REGION Network 54: CM Vision Z Axis Command posAbsolute
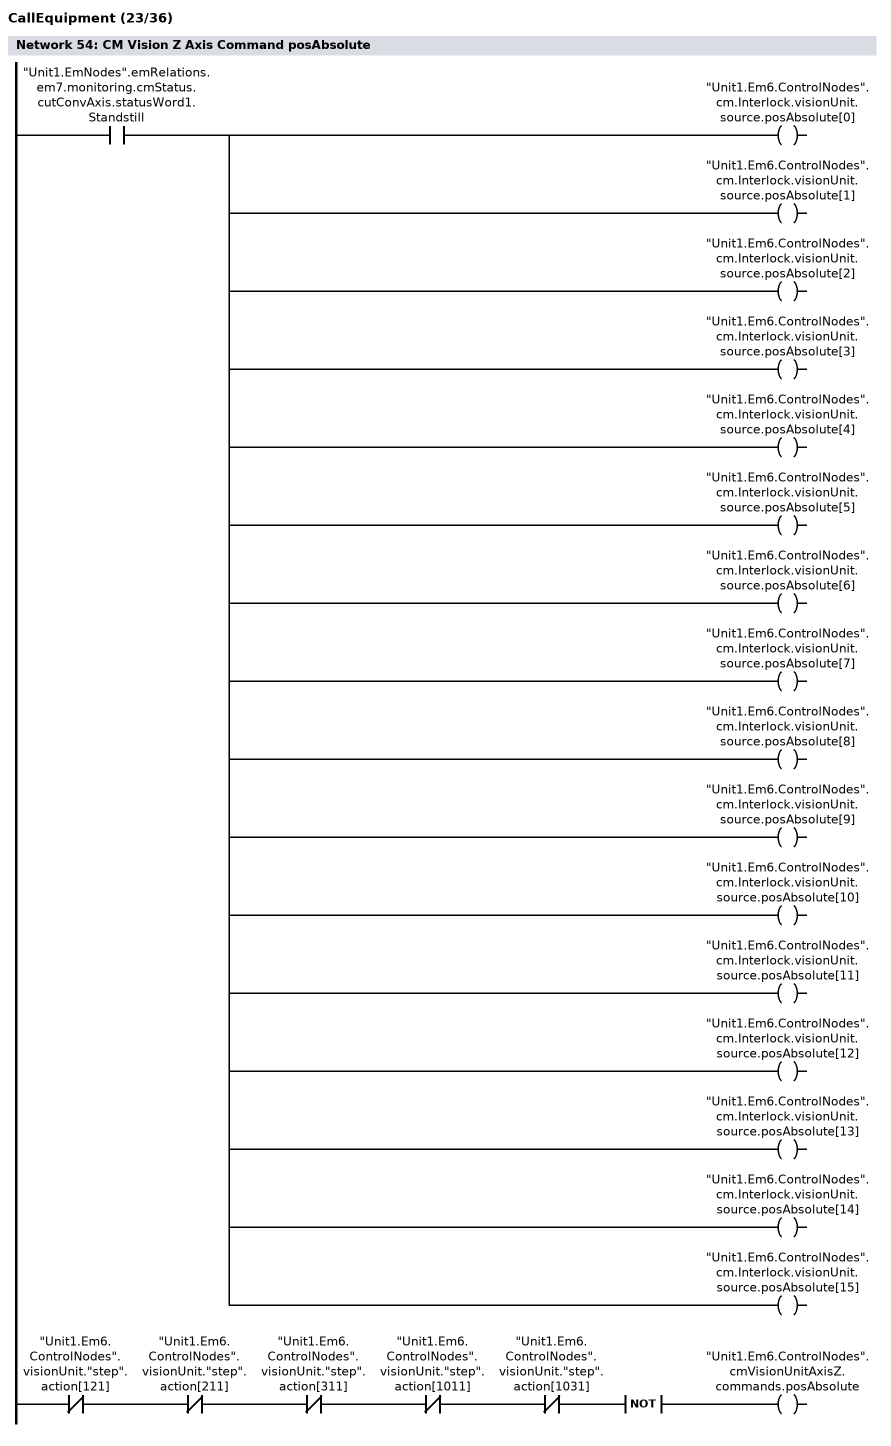
   RUNG wire#powerrail
      Contact( "Unit1.EmNodes".emRelations.em7.monitoring.cmStatus.cutConvAxis.statusWord1.Standstill )
      wire#w1
      Coil( "Unit1.Em6.ControlNodes".cm.Interlock.visionUnit.source.posAbsolute[0] )
   END_RUNG
   RUNG wire#w1
      Coil( "Unit1.Em6.ControlNodes".cm.Interlock.visionUnit.source.posAbsolute[1] )
   END_RUNG
   RUNG wire#w1
      Coil( "Unit1.Em6.ControlNodes".cm.Interlock.visionUnit.source.posAbsolute[2] )
   END_RUNG
   RUNG wire#w1
      Coil( "Unit1.Em6.ControlNodes".cm.Interlock.visionUnit.source.posAbsolute[3] )
   END_RUNG
   RUNG wire#w1
      Coil( "Unit1.Em6.ControlNodes".cm.Interlock.visionUnit.source.posAbsolute[4] )
   END_RUNG
   RUNG wire#w1
      Coil( "Unit1.Em6.ControlNodes".cm.Interlock.visionUnit.source.posAbsolute[5] )
   END_RUNG
   RUNG wire#w1
      Coil( "Unit1.Em6.ControlNodes".cm.Interlock.visionUnit.source.posAbsolute[6] )
   END_RUNG
   RUNG wire#w1
      Coil( "Unit1.Em6.ControlNodes".cm.Interlock.visionUnit.source.posAbsolute[7] )
   END_RUNG
   RUNG wire#w1
      Coil( "Unit1.Em6.ControlNodes".cm.Interlock.visionUnit.source.posAbsolute[8] )
   END_RUNG
   RUNG wire#w1
      Coil( "Unit1.Em6.ControlNodes".cm.Interlock.visionUnit.source.posAbsolute[9] )
   END_RUNG
   RUNG wire#w1
      Coil( "Unit1.Em6.ControlNodes".cm.Interlock.visionUnit.source.posAbsolute[10] )
   END_RUNG
   RUNG wire#w1
      Coil( "Unit1.Em6.ControlNodes".cm.Interlock.visionUnit.source.posAbsolute[11] )
   END_RUNG
   RUNG wire#w1
      Coil( "Unit1.Em6.ControlNodes".cm.Interlock.visionUnit.source.posAbsolute[12] )
   END_RUNG
   RUNG wire#w1
      Coil( "Unit1.Em6.ControlNodes".cm.Interlock.visionUnit.source.posAbsolute[13] )
   END_RUNG
   RUNG wire#w1
      Coil( "Unit1.Em6.ControlNodes".cm.Interlock.visionUnit.source.posAbsolute[14] )
   END_RUNG
   RUNG wire#w1
      Coil( "Unit1.Em6.ControlNodes".cm.Interlock.visionUnit.source.posAbsolute[15] )
   END_RUNG
   RUNG wire#powerrail
      I_Contact( "Unit1.Em6.ControlNodes".visionUnit."step".action[121] )
      I_Contact( "Unit1.Em6.ControlNodes".visionUnit."step".action[211] )
      I_Contact( "Unit1.Em6.ControlNodes".visionUnit."step".action[311] )
      I_Contact( "Unit1.Em6.ControlNodes".visionUnit."step".action[1011] )
      I_Contact( "Unit1.Em6.ControlNodes".visionUnit."step".action[1031] )
      Not()
      Coil( "Unit1.Em6.ControlNodes".cmVisionUnitAxisZ.commands.posAbsolute )
   END_RUNG
   // the same network as SCL:
   "Unit1.Em6.ControlNodes".cm.Interlock.visionUnit.source.posAbsolute[0] := "Unit1.EmNodes".emRelations.em7.monitoring.cmStatus.cutConvAxis.statusWord1.Standstill;
   "Unit1.Em6.ControlNodes".cm.Interlock.visionUnit.source.posAbsolute[1] := "Unit1.EmNodes".emRelations.em7.monitoring.cmStatus.cutConvAxis.statusWord1.Standstill;
   "Unit1.Em6.ControlNodes".cm.Interlock.visionUnit.source.posAbsolute[2] := "Unit1.EmNodes".emRelations.em7.monitoring.cmStatus.cutConvAxis.statusWord1.Standstill;
   "Unit1.Em6.ControlNodes".cm.Interlock.visionUnit.source.posAbsolute[3] := "Unit1.EmNodes".emRelations.em7.monitoring.cmStatus.cutConvAxis.statusWord1.Standstill;
   "Unit1.Em6.ControlNodes".cm.Interlock.visionUnit.source.posAbsolute[4] := "Unit1.EmNodes".emRelations.em7.monitoring.cmStatus.cutConvAxis.statusWord1.Standstill;
   "Unit1.Em6.ControlNodes".cm.Interlock.visionUnit.source.posAbsolute[5] := "Unit1.EmNodes".emRelations.em7.monitoring.cmStatus.cutConvAxis.statusWord1.Standstill;
   "Unit1.Em6.ControlNodes".cm.Interlock.visionUnit.source.posAbsolute[6] := "Unit1.EmNodes".emRelations.em7.monitoring.cmStatus.cutConvAxis.statusWord1.Standstill;
   "Unit1.Em6.ControlNodes".cm.Interlock.visionUnit.source.posAbsolute[7] := "Unit1.EmNodes".emRelations.em7.monitoring.cmStatus.cutConvAxis.statusWord1.Standstill;
   "Unit1.Em6.ControlNodes".cm.Interlock.visionUnit.source.posAbsolute[8] := "Unit1.EmNodes".emRelations.em7.monitoring.cmStatus.cutConvAxis.statusWord1.Standstill;
   "Unit1.Em6.ControlNodes".cm.Interlock.visionUnit.source.posAbsolute[9] := "Unit1.EmNodes".emRelations.em7.monitoring.cmStatus.cutConvAxis.statusWord1.Standstill;
   "Unit1.Em6.ControlNodes".cm.Interlock.visionUnit.source.posAbsolute[10] := "Unit1.EmNodes".emRelations.em7.monitoring.cmStatus.cutConvAxis.statusWord1.Standstill;
   "Unit1.Em6.ControlNodes".cm.Interlock.visionUnit.source.posAbsolute[11] := "Unit1.EmNodes".emRelations.em7.monitoring.cmStatus.cutConvAxis.statusWord1.Standstill;
   "Unit1.Em6.ControlNodes".cm.Interlock.visionUnit.source.posAbsolute[12] := "Unit1.EmNodes".emRelations.em7.monitoring.cmStatus.cutConvAxis.statusWord1.Standstill;
   "Unit1.Em6.ControlNodes".cm.Interlock.visionUnit.source.posAbsolute[13] := "Unit1.EmNodes".emRelations.em7.monitoring.cmStatus.cutConvAxis.statusWord1.Standstill;
   "Unit1.Em6.ControlNodes".cm.Interlock.visionUnit.source.posAbsolute[14] := "Unit1.EmNodes".emRelations.em7.monitoring.cmStatus.cutConvAxis.statusWord1.Standstill;
   "Unit1.Em6.ControlNodes".cm.Interlock.visionUnit.source.posAbsolute[15] := "Unit1.EmNodes".emRelations.em7.monitoring.cmStatus.cutConvAxis.statusWord1.Standstill;
   "Unit1.Em6.ControlNodes".cmVisionUnitAxisZ.commands.posAbsolute := NOT (NOT "Unit1.Em6.ControlNodes".visionUnit."step".action[121] AND NOT "Unit1.Em6.ControlNodes".visionUnit."step".action[211] AND NOT "Unit1.Em6.ControlNodes".visionUnit."step".action[311] AND NOT "Unit1.Em6.ControlNodes".visionUnit."step".action[1011] AND NOT "Unit1.Em6.ControlNodes".visionUnit."step".action[1031]);
END_REGION

REGION Network 55: Call CM Vision Z Axis (LER_Interlock Summary)
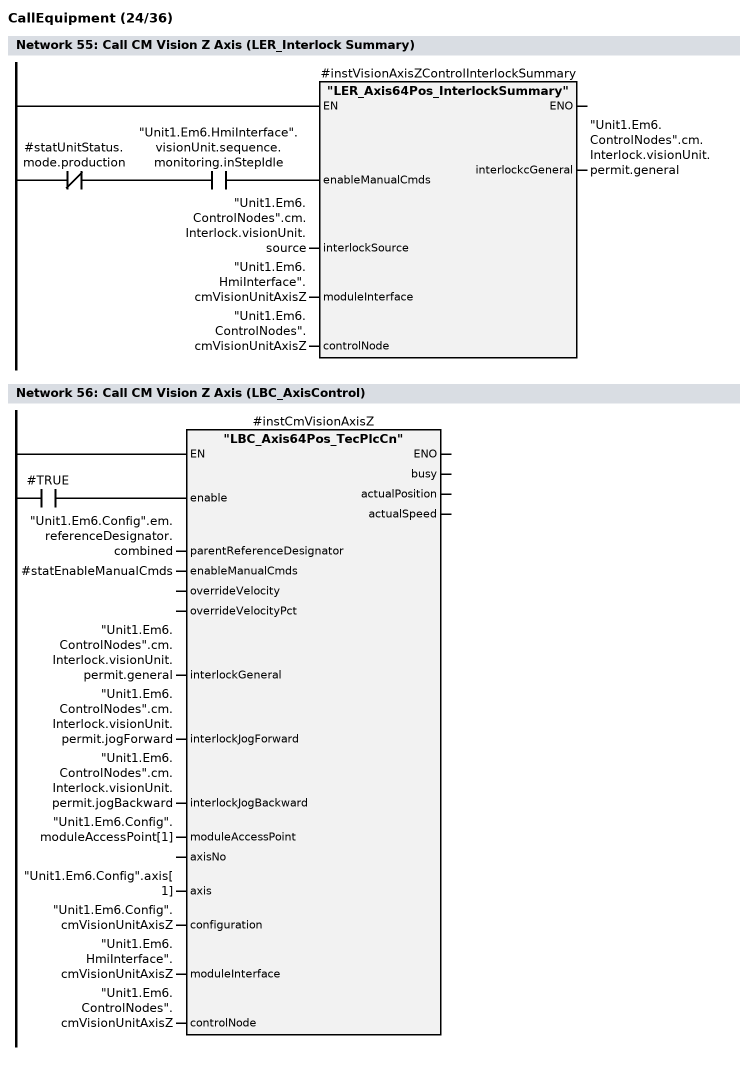
   RUNG wire#powerrail
      #instVisionAxisZControlInterlockSummary(enableManualCmds := wire#w1, interlockSource := "Unit1.Em6.ControlNodes".cm.Interlock.visionUnit.source, moduleInterface := "Unit1.Em6.HmiInterface".cmVisionUnitAxisZ, controlNode := "Unit1.Em6.ControlNodes".cmVisionUnitAxisZ, interlockcGeneral => "Unit1.Em6.ControlNodes".cm.Interlock.visionUnit.permit.general)
   END_RUNG
   RUNG wire#powerrail
      I_Contact( #statUnitStatus.mode.production )
      Contact( "Unit1.Em6.HmiInterface".visionUnit.sequence.monitoring.inStepIdle )
   END_RUNG wire#w1
   // the same network as SCL:
   #instVisionAxisZControlInterlockSummary(enableManualCmds := NOT #statUnitStatus.mode.production AND "Unit1.Em6.HmiInterface".visionUnit.sequence.monitoring.inStepIdle,   // "LER_Axis64Pos_InterlockSummary"
                           interlockSource := "Unit1.Em6.ControlNodes".cm.Interlock.visionUnit.source,
                           moduleInterface := "Unit1.Em6.HmiInterface".cmVisionUnitAxisZ,
                           controlNode := "Unit1.Em6.ControlNodes".cmVisionUnitAxisZ,
                           interlockcGeneral => "Unit1.Em6.ControlNodes".cm.Interlock.visionUnit.permit.general);
END_REGION

REGION Network 56: Call CM Vision Z Axis (LBC_AxisControl)
   RUNG wire#powerrail
      #instCmVisionAxisZ(enable := wire#w1, parentReferenceDesignator := "Unit1.Em6.Config".em.referenceDesignator.combined, enableManualCmds := #statEnableManualCmds, overrideVelocity :=, overrideVelocityPct :=, interlockGeneral := "Unit1.Em6.ControlNodes".cm.Interlock.visionUnit.permit.general, interlockJogForward := "Unit1.Em6.ControlNodes".cm.Interlock.visionUnit.permit.jogForward, interlockJogBackward := "Unit1.Em6.ControlNodes".cm.Interlock.visionUnit.permit.jogBackward, moduleAccessPoint := "Unit1.Em6.Config".moduleAccessPoint[1], axisNo :=, axis := "Unit1.Em6.Config".axis[1], configuration := "Unit1.Em6.Config".cmVisionUnitAxisZ, moduleInterface := "Unit1.Em6.HmiInterface".cmVisionUnitAxisZ, controlNode := "Unit1.Em6.ControlNodes".cmVisionUnitAxisZ, busy =>, actualPosition =>, actualSpeed =>)
   END_RUNG
   RUNG wire#powerrail
      Contact( #TRUE )
   END_RUNG wire#w1
   // the same network as SCL:
   #instCmVisionAxisZ(enable := #TRUE,   // "LBC_Axis64Pos_TecPlcCn"
                      parentReferenceDesignator := "Unit1.Em6.Config".em.referenceDesignator.combined,
                      enableManualCmds := #statEnableManualCmds,
                      interlockGeneral := "Unit1.Em6.ControlNodes".cm.Interlock.visionUnit.permit.general,
                      interlockJogForward := "Unit1.Em6.ControlNodes".cm.Interlock.visionUnit.permit.jogForward,
                      interlockJogBackward := "Unit1.Em6.ControlNodes".cm.Interlock.visionUnit.permit.jogBackward,
                      moduleAccessPoint := "Unit1.Em6.Config".moduleAccessPoint[1],
                      axis := "Unit1.Em6.Config".axis[1],
                      configuration := "Unit1.Em6.Config".cmVisionUnitAxisZ,
                      moduleInterface := "Unit1.Em6.HmiInterface".cmVisionUnitAxisZ,
                      controlNode := "Unit1.Em6.ControlNodes".cmVisionUnitAxisZ);
END_REGION

REGION Network 57: Call CM Vision Z Axis (LER_ServoTorqueCal)
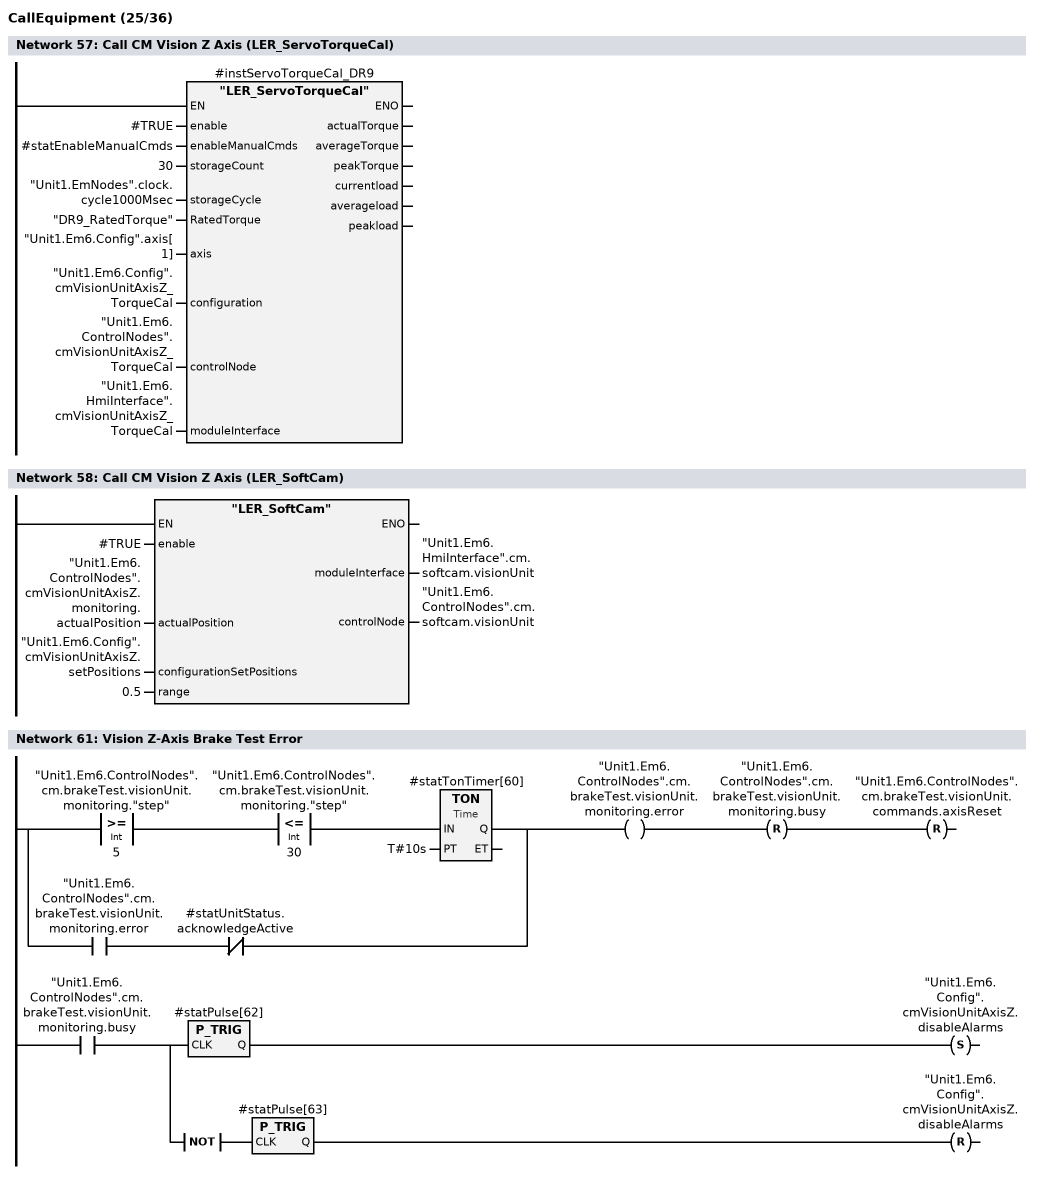
   RUNG wire#powerrail
      #instServoTorqueCal_DR9(enable := #TRUE, enableManualCmds := #statEnableManualCmds, storageCount := 30, storageCycle := "Unit1.EmNodes".clock.cycle1000Msec, RatedTorque := "DR9_RatedTorque", axis := "Unit1.Em6.Config".axis[1], configuration := "Unit1.Em6.Config".cmVisionUnitAxisZ_TorqueCal, controlNode := "Unit1.Em6.ControlNodes".cmVisionUnitAxisZ_TorqueCal, moduleInterface := "Unit1.Em6.HmiInterface".cmVisionUnitAxisZ_TorqueCal, actualTorque =>, averageTorque =>, peakTorque =>, currentload =>, averageload =>, peakload =>)
   END_RUNG
   // the same network as SCL:
   #instServoTorqueCal_DR9(enable := #TRUE,   // "LER_ServoTorqueCal"
                           enableManualCmds := #statEnableManualCmds,
                           storageCount := 30,
                           storageCycle := "Unit1.EmNodes".clock.cycle1000Msec,
                           RatedTorque := "DR9_RatedTorque",
                           axis := "Unit1.Em6.Config".axis[1],
                           configuration := "Unit1.Em6.Config".cmVisionUnitAxisZ_TorqueCal,
                           controlNode := "Unit1.Em6.ControlNodes".cmVisionUnitAxisZ_TorqueCal,
                           moduleInterface := "Unit1.Em6.HmiInterface".cmVisionUnitAxisZ_TorqueCal);
END_REGION

REGION Network 58: Call CM Vision Z Axis (LER_SoftCam)
   RUNG wire#powerrail
      "LER_SoftCam"(enable := #TRUE, actualPosition := "Unit1.Em6.ControlNodes".cmVisionUnitAxisZ.monitoring.actualPosition, configurationSetPositions := "Unit1.Em6.Config".cmVisionUnitAxisZ.setPositions, range := 0.5, moduleInterface => "Unit1.Em6.HmiInterface".cm.softcam.visionUnit, controlNode => "Unit1.Em6.ControlNodes".cm.softcam.visionUnit)
   END_RUNG
   // the same network as SCL:
   "LER_SoftCam"(enable := #TRUE,
                 actualPosition := "Unit1.Em6.ControlNodes".cmVisionUnitAxisZ.monitoring.actualPosition,
                 configurationSetPositions := "Unit1.Em6.Config".cmVisionUnitAxisZ.setPositions,
                 range := 0.5,
                 moduleInterface => "Unit1.Em6.HmiInterface".cm.softcam.visionUnit,
                 controlNode => "Unit1.Em6.ControlNodes".cm.softcam.visionUnit);
END_REGION

REGION Network 60: ******************** Brake Test (Axis) ********************
END_REGION

REGION Network 61: Vision Z-Axis Brake Test Error
   RUNG wire#powerrail
      { S7_Templates := "SrcType := Int" } GE_Contact(in1 := "Unit1.Em6.ControlNodes".cm.brakeTest.visionUnit.monitoring."step", in2 := 5)
      { S7_Templates := "SrcType := Int" } LE_Contact(in1 := "Unit1.Em6.ControlNodes".cm.brakeTest.visionUnit.monitoring."step", in2 := 30)
      { S7_Templates := "time_type := Time" } #statTonTimer[60].TON(pt := T#10s, et =>)
      wire#w1
      Coil( "Unit1.Em6.ControlNodes".cm.brakeTest.visionUnit.monitoring.error )
      R_Coil( "Unit1.Em6.ControlNodes".cm.brakeTest.visionUnit.monitoring.busy )
      R_Coil( "Unit1.Em6.ControlNodes".cm.brakeTest.visionUnit.commands.axisReset )
   END_RUNG
   RUNG wire#powerrail
      Contact( "Unit1.Em6.ControlNodes".cm.brakeTest.visionUnit.monitoring.error )
      I_Contact( #statUnitStatus.acknowledgeActive )
   END_RUNG wire#w1
   RUNG wire#powerrail
      Contact( "Unit1.Em6.ControlNodes".cm.brakeTest.visionUnit.monitoring.busy )
      wire#w2
      P_Trig( #statPulse[62] )
      S_Coil( "Unit1.Em6.Config".cmVisionUnitAxisZ.disableAlarms )
   END_RUNG
   RUNG wire#w2
      Not()
      P_Trig( #statPulse[63] )
      R_Coil( "Unit1.Em6.Config".cmVisionUnitAxisZ.disableAlarms )
   END_RUNG
   // the same network as SCL:
   #statTonTimer[60].TON(IN := ("Unit1.Em6.ControlNodes".cm.brakeTest.visionUnit.monitoring."step" >= 5) AND ("Unit1.Em6.ControlNodes".cm.brakeTest.visionUnit.monitoring."step" <= 30),
                         PT := T#10s);
   "Unit1.Em6.ControlNodes".cm.brakeTest.visionUnit.monitoring.error := #statTonTimer[60].Q OR ("Unit1.Em6.ControlNodes".cm.brakeTest.visionUnit.monitoring.error AND NOT #statUnitStatus.acknowledgeActive);
   IF "Unit1.Em6.ControlNodes".cm.brakeTest.visionUnit.monitoring.error THEN
       "Unit1.Em6.ControlNodes".cm.brakeTest.visionUnit.monitoring.busy := FALSE;
       "Unit1.Em6.ControlNodes".cm.brakeTest.visionUnit.commands.axisReset := FALSE;
   END_IF;
   #_w1 := "Unit1.Em6.ControlNodes".cm.brakeTest.visionUnit.monitoring.busy AND NOT #statPulse[62];   // rising edge
   #statPulse[62] := "Unit1.Em6.ControlNodes".cm.brakeTest.visionUnit.monitoring.busy;
   IF #_w1 THEN "Unit1.Em6.Config".cmVisionUnitAxisZ.disableAlarms := TRUE; END_IF;
   #_w2 := NOT "Unit1.Em6.ControlNodes".cm.brakeTest.visionUnit.monitoring.busy AND NOT #statPulse[63];   // rising edge
   #statPulse[63] := NOT "Unit1.Em6.ControlNodes".cm.brakeTest.visionUnit.monitoring.busy;
   IF #_w2 THEN "Unit1.Em6.Config".cmVisionUnitAxisZ.disableAlarms := FALSE; END_IF;
END_REGION

REGION Network 62: Vision Z-Axis Brake Test Initialize
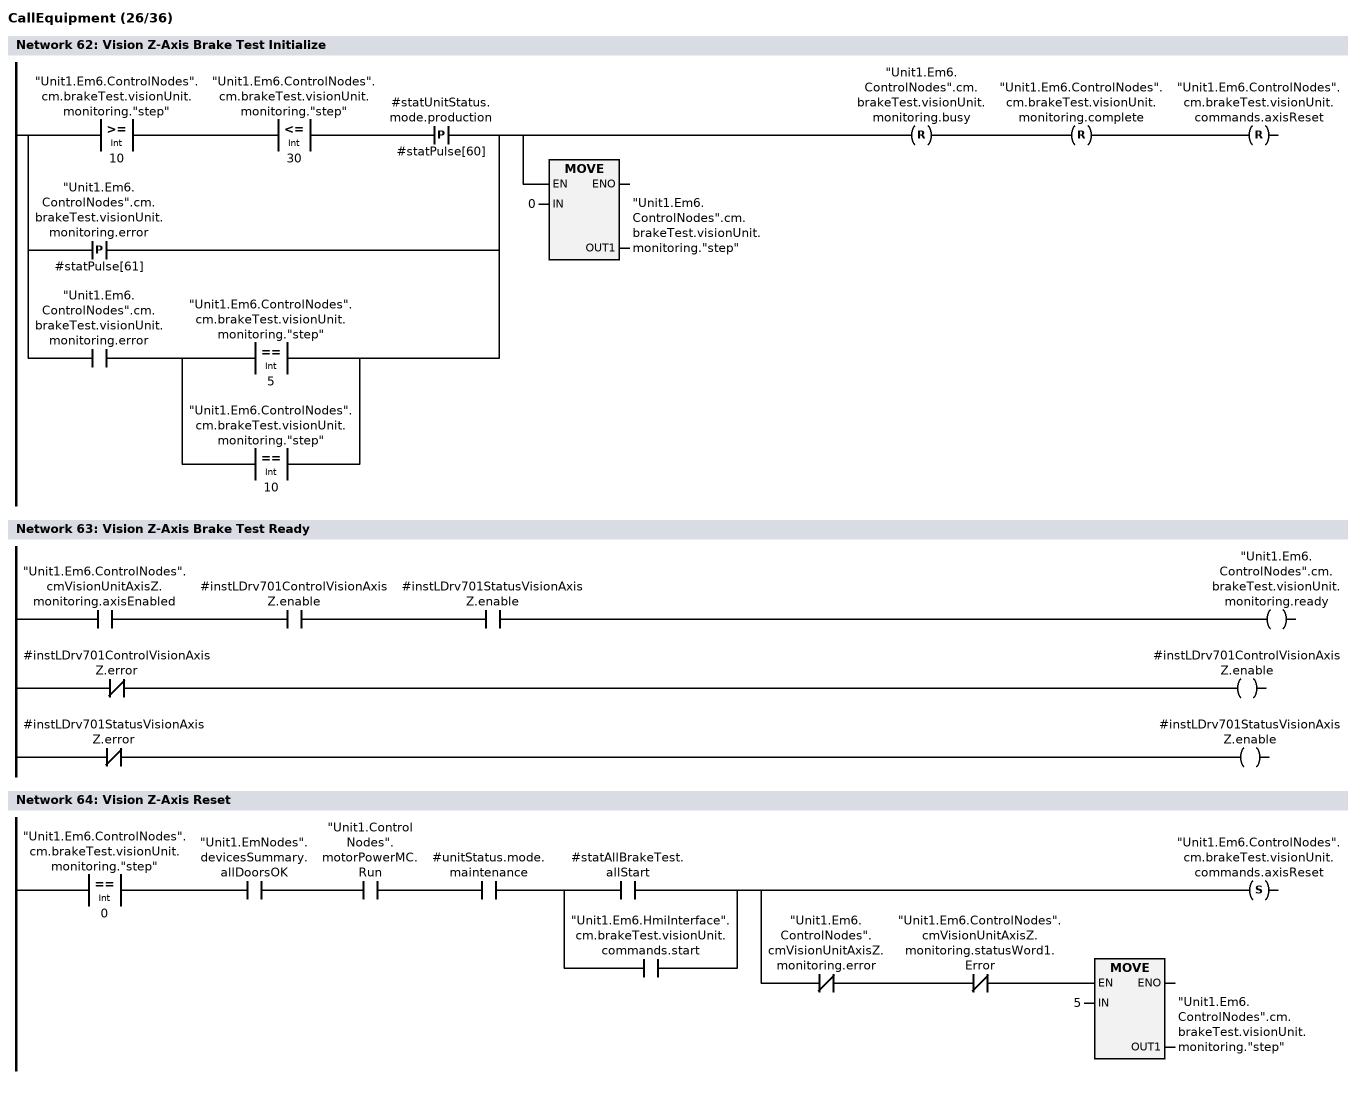
   RUNG wire#powerrail
      { S7_Templates := "SrcType := Int" } GE_Contact(in1 := "Unit1.Em6.ControlNodes".cm.brakeTest.visionUnit.monitoring."step", in2 := 10)
      { S7_Templates := "SrcType := Int" } LE_Contact(in1 := "Unit1.Em6.ControlNodes".cm.brakeTest.visionUnit.monitoring."step", in2 := 30)
      P_Contact(operand := #statUnitStatus.mode.production, bit := #statPulse[60])
      wire#w1
      R_Coil( "Unit1.Em6.ControlNodes".cm.brakeTest.visionUnit.monitoring.busy )
      R_Coil( "Unit1.Em6.ControlNodes".cm.brakeTest.visionUnit.monitoring.complete )
      R_Coil( "Unit1.Em6.ControlNodes".cm.brakeTest.visionUnit.commands.axisReset )
   END_RUNG
   RUNG wire#powerrail
      P_Contact(operand := "Unit1.Em6.ControlNodes".cm.brakeTest.visionUnit.monitoring.error, bit := #statPulse[61])
   END_RUNG wire#w1
   RUNG wire#powerrail
      Contact( "Unit1.Em6.ControlNodes".cm.brakeTest.visionUnit.monitoring.error )
      wire#w2
      { S7_Templates := "SrcType := Int" } EQ_Contact(in1 := "Unit1.Em6.ControlNodes".cm.brakeTest.visionUnit.monitoring."step", in2 := 5)
   END_RUNG wire#w1
   RUNG wire#w2
      { S7_Templates := "SrcType := Int" } EQ_Contact(in1 := "Unit1.Em6.ControlNodes".cm.brakeTest.visionUnit.monitoring."step", in2 := 10)
   END_RUNG wire#w1
   RUNG wire#w1
      Move(in := 0, out1 => "Unit1.Em6.ControlNodes".cm.brakeTest.visionUnit.monitoring."step")
   END_RUNG
   // the same network as SCL:
   #_w1 := ("Unit1.Em6.ControlNodes".cm.brakeTest.visionUnit.monitoring."step" >= 10) AND ("Unit1.Em6.ControlNodes".cm.brakeTest.visionUnit.monitoring."step" <= 30) AND #statUnitStatus.mode.production AND NOT #statPulse[60];   // rising edge of #statUnitStatus.mode.production
   #statPulse[60] := #statUnitStatus.mode.production;
   #_w2 := "Unit1.Em6.ControlNodes".cm.brakeTest.visionUnit.monitoring.error AND NOT #statPulse[61];   // rising edge of "Unit1.Em6.ControlNodes".cm.brakeTest.visionUnit.monitoring.error
   #statPulse[61] := "Unit1.Em6.ControlNodes".cm.brakeTest.visionUnit.monitoring.error;
   IF #_w1 OR #_w2 OR ("Unit1.Em6.ControlNodes".cm.brakeTest.visionUnit.monitoring.error AND (("Unit1.Em6.ControlNodes".cm.brakeTest.visionUnit.monitoring."step" = 5) OR ("Unit1.Em6.ControlNodes".cm.brakeTest.visionUnit.monitoring."step" = 10))) THEN
       "Unit1.Em6.ControlNodes".cm.brakeTest.visionUnit.monitoring.busy := FALSE;
       "Unit1.Em6.ControlNodes".cm.brakeTest.visionUnit.monitoring.complete := FALSE;
       "Unit1.Em6.ControlNodes".cm.brakeTest.visionUnit.commands.axisReset := FALSE;
       "Unit1.Em6.ControlNodes".cm.brakeTest.visionUnit.monitoring."step" := 0;
   END_IF;
END_REGION

REGION Network 63: Vision Z-Axis Brake Test Ready
   RUNG wire#powerrail
      Contact( "Unit1.Em6.ControlNodes".cmVisionUnitAxisZ.monitoring.axisEnabled )
      Contact( #instLDrv701ControlVisionAxisZ.enable )
      Contact( #instLDrv701StatusVisionAxisZ.enable )
      Coil( "Unit1.Em6.ControlNodes".cm.brakeTest.visionUnit.monitoring.ready )
   END_RUNG
   RUNG wire#powerrail
      I_Contact( #instLDrv701ControlVisionAxisZ.error )
      Coil( #instLDrv701ControlVisionAxisZ.enable )
   END_RUNG
   RUNG wire#powerrail
      I_Contact( #instLDrv701StatusVisionAxisZ.error )
      Coil( #instLDrv701StatusVisionAxisZ.enable )
   END_RUNG
   // the same network as SCL:
   "Unit1.Em6.ControlNodes".cm.brakeTest.visionUnit.monitoring.ready := "Unit1.Em6.ControlNodes".cmVisionUnitAxisZ.monitoring.axisEnabled AND #instLDrv701ControlVisionAxisZ.enable AND #instLDrv701StatusVisionAxisZ.enable;
   #instLDrv701ControlVisionAxisZ.enable := NOT #instLDrv701ControlVisionAxisZ.error;
   #instLDrv701StatusVisionAxisZ.enable := NOT #instLDrv701StatusVisionAxisZ.error;
END_REGION

REGION Network 64: Vision Z-Axis Reset
   RUNG wire#powerrail
      { S7_Templates := "SrcType := Int" } EQ_Contact(in1 := "Unit1.Em6.ControlNodes".cm.brakeTest.visionUnit.monitoring."step", in2 := 0)
      Contact( "Unit1.EmNodes".devicesSummary.allDoorsOK )
      Contact( "Unit1.ControlNodes".motorPowerMC.Run )
      Contact( #unitStatus.mode.maintenance )
      wire#w1
      Contact( #statAllBrakeTest.allStart )
      wire#w2
      S_Coil( "Unit1.Em6.ControlNodes".cm.brakeTest.visionUnit.commands.axisReset )
   END_RUNG
   RUNG wire#w1
      Contact( "Unit1.Em6.HmiInterface".cm.brakeTest.visionUnit.commands.start )
   END_RUNG wire#w2
   RUNG wire#w2
      I_Contact( "Unit1.Em6.ControlNodes".cmVisionUnitAxisZ.monitoring.error )
      I_Contact( "Unit1.Em6.ControlNodes".cmVisionUnitAxisZ.monitoring.statusWord1.Error )
      Move(in := 5, out1 => "Unit1.Em6.ControlNodes".cm.brakeTest.visionUnit.monitoring."step")
   END_RUNG
   // the same network as SCL:
   #_w1 := ("Unit1.Em6.ControlNodes".cm.brakeTest.visionUnit.monitoring."step" = 0) AND "Unit1.EmNodes".devicesSummary.allDoorsOK AND "Unit1.ControlNodes".motorPowerMC.Run AND #unitStatus.mode.maintenance AND (#statAllBrakeTest.allStart OR "Unit1.Em6.HmiInterface".cm.brakeTest.visionUnit.commands.start);
   IF #_w1 THEN "Unit1.Em6.ControlNodes".cm.brakeTest.visionUnit.commands.axisReset := TRUE; END_IF;
   IF #_w1 AND NOT "Unit1.Em6.ControlNodes".cmVisionUnitAxisZ.monitoring.error AND NOT "Unit1.Em6.ControlNodes".cmVisionUnitAxisZ.monitoring.statusWord1.Error THEN
       "Unit1.Em6.ControlNodes".cm.brakeTest.visionUnit.monitoring."step" := 5;
   END_IF;
END_REGION

REGION Network 65: Vision Z-Axis Brake Test Commands
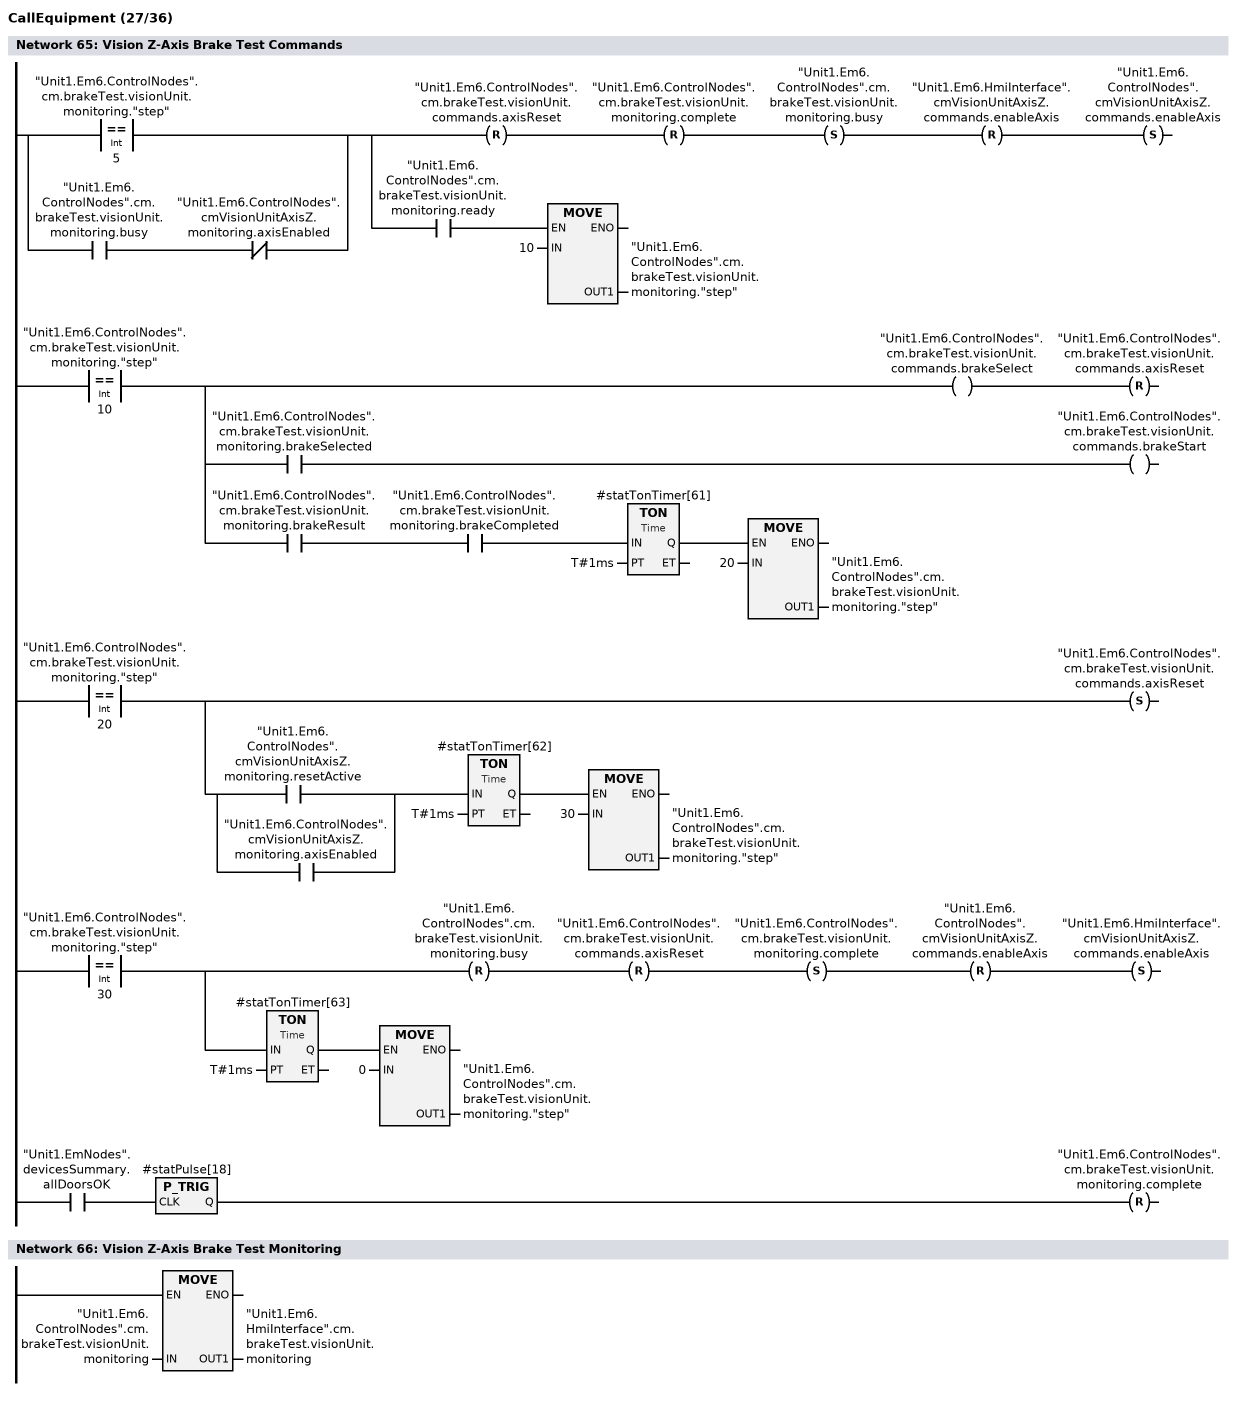
   RUNG wire#powerrail
      { S7_Templates := "SrcType := Int" } EQ_Contact(in1 := "Unit1.Em6.ControlNodes".cm.brakeTest.visionUnit.monitoring."step", in2 := 5)
      wire#w1
      R_Coil( "Unit1.Em6.ControlNodes".cm.brakeTest.visionUnit.commands.axisReset )
      R_Coil( "Unit1.Em6.ControlNodes".cm.brakeTest.visionUnit.monitoring.complete )
      S_Coil( "Unit1.Em6.ControlNodes".cm.brakeTest.visionUnit.monitoring.busy )
      R_Coil( "Unit1.Em6.HmiInterface".cmVisionUnitAxisZ.commands.enableAxis )
      S_Coil( "Unit1.Em6.ControlNodes".cmVisionUnitAxisZ.commands.enableAxis )
   END_RUNG
   RUNG wire#powerrail
      Contact( "Unit1.Em6.ControlNodes".cm.brakeTest.visionUnit.monitoring.busy )
      I_Contact( "Unit1.Em6.ControlNodes".cmVisionUnitAxisZ.monitoring.axisEnabled )
   END_RUNG wire#w1
   RUNG wire#w1
      Contact( "Unit1.Em6.ControlNodes".cm.brakeTest.visionUnit.monitoring.ready )
      Move(in := 10, out1 => "Unit1.Em6.ControlNodes".cm.brakeTest.visionUnit.monitoring."step")
   END_RUNG
   RUNG wire#powerrail
      { S7_Templates := "SrcType := Int" } EQ_Contact(in1 := "Unit1.Em6.ControlNodes".cm.brakeTest.visionUnit.monitoring."step", in2 := 10)
      wire#w2
      Coil( "Unit1.Em6.ControlNodes".cm.brakeTest.visionUnit.commands.brakeSelect )
      R_Coil( "Unit1.Em6.ControlNodes".cm.brakeTest.visionUnit.commands.axisReset )
   END_RUNG
   RUNG wire#w2
      Contact( "Unit1.Em6.ControlNodes".cm.brakeTest.visionUnit.monitoring.brakeSelected )
      Coil( "Unit1.Em6.ControlNodes".cm.brakeTest.visionUnit.commands.brakeStart )
   END_RUNG
   RUNG wire#w2
      Contact( "Unit1.Em6.ControlNodes".cm.brakeTest.visionUnit.monitoring.brakeResult )
      Contact( "Unit1.Em6.ControlNodes".cm.brakeTest.visionUnit.monitoring.brakeCompleted )
      { S7_Templates := "time_type := Time" } #statTonTimer[61].TON(pt := T#1ms, et =>)
      Move(in := 20, out1 => "Unit1.Em6.ControlNodes".cm.brakeTest.visionUnit.monitoring."step")
   END_RUNG
   RUNG wire#powerrail
      { S7_Templates := "SrcType := Int" } EQ_Contact(in1 := "Unit1.Em6.ControlNodes".cm.brakeTest.visionUnit.monitoring."step", in2 := 20)
      wire#w3
      S_Coil( "Unit1.Em6.ControlNodes".cm.brakeTest.visionUnit.commands.axisReset )
   END_RUNG
   RUNG wire#w3
      Contact( "Unit1.Em6.ControlNodes".cmVisionUnitAxisZ.monitoring.resetActive )
      wire#w4
      { S7_Templates := "time_type := Time" } #statTonTimer[62].TON(pt := T#1ms, et =>)
      Move(in := 30, out1 => "Unit1.Em6.ControlNodes".cm.brakeTest.visionUnit.monitoring."step")
   END_RUNG
   RUNG wire#w3
      Contact( "Unit1.Em6.ControlNodes".cmVisionUnitAxisZ.monitoring.axisEnabled )
   END_RUNG wire#w4
   RUNG wire#powerrail
      { S7_Templates := "SrcType := Int" } EQ_Contact(in1 := "Unit1.Em6.ControlNodes".cm.brakeTest.visionUnit.monitoring."step", in2 := 30)
      wire#w5
      R_Coil( "Unit1.Em6.ControlNodes".cm.brakeTest.visionUnit.monitoring.busy )
      R_Coil( "Unit1.Em6.ControlNodes".cm.brakeTest.visionUnit.commands.axisReset )
      S_Coil( "Unit1.Em6.ControlNodes".cm.brakeTest.visionUnit.monitoring.complete )
      R_Coil( "Unit1.Em6.ControlNodes".cmVisionUnitAxisZ.commands.enableAxis )
      S_Coil( "Unit1.Em6.HmiInterface".cmVisionUnitAxisZ.commands.enableAxis )
   END_RUNG
   RUNG wire#w5
      { S7_Templates := "time_type := Time" } #statTonTimer[63].TON(pt := T#1ms, et =>)
      Move(in := 0, out1 => "Unit1.Em6.ControlNodes".cm.brakeTest.visionUnit.monitoring."step")
   END_RUNG
   RUNG wire#powerrail
      Contact( "Unit1.EmNodes".devicesSummary.allDoorsOK )
      P_Trig( #statPulse[18] )
      R_Coil( "Unit1.Em6.ControlNodes".cm.brakeTest.visionUnit.monitoring.complete )
   END_RUNG
   // the same network as SCL:
   #_w1 := ("Unit1.Em6.ControlNodes".cm.brakeTest.visionUnit.monitoring."step" = 5) OR ("Unit1.Em6.ControlNodes".cm.brakeTest.visionUnit.monitoring.busy AND NOT "Unit1.Em6.ControlNodes".cmVisionUnitAxisZ.monitoring.axisEnabled);
   IF #_w1 THEN
       "Unit1.Em6.ControlNodes".cm.brakeTest.visionUnit.commands.axisReset := FALSE;
       "Unit1.Em6.ControlNodes".cm.brakeTest.visionUnit.monitoring.complete := FALSE;
       "Unit1.Em6.ControlNodes".cm.brakeTest.visionUnit.monitoring.busy := TRUE;
       "Unit1.Em6.HmiInterface".cmVisionUnitAxisZ.commands.enableAxis := FALSE;
       "Unit1.Em6.ControlNodes".cmVisionUnitAxisZ.commands.enableAxis := TRUE;
   END_IF;
   IF #_w1 AND "Unit1.Em6.ControlNodes".cm.brakeTest.visionUnit.monitoring.ready THEN
       "Unit1.Em6.ControlNodes".cm.brakeTest.visionUnit.monitoring."step" := 10;
   END_IF;
   "Unit1.Em6.ControlNodes".cm.brakeTest.visionUnit.commands.brakeSelect := "Unit1.Em6.ControlNodes".cm.brakeTest.visionUnit.monitoring."step" = 10;
   IF "Unit1.Em6.ControlNodes".cm.brakeTest.visionUnit.commands.brakeSelect THEN
       "Unit1.Em6.ControlNodes".cm.brakeTest.visionUnit.commands.axisReset := FALSE;
   END_IF;
   "Unit1.Em6.ControlNodes".cm.brakeTest.visionUnit.commands.brakeStart := "Unit1.Em6.ControlNodes".cm.brakeTest.visionUnit.commands.brakeSelect AND "Unit1.Em6.ControlNodes".cm.brakeTest.visionUnit.monitoring.brakeSelected;
   #statTonTimer[61].TON(IN := "Unit1.Em6.ControlNodes".cm.brakeTest.visionUnit.commands.brakeSelect AND "Unit1.Em6.ControlNodes".cm.brakeTest.visionUnit.monitoring.brakeResult AND "Unit1.Em6.ControlNodes".cm.brakeTest.visionUnit.monitoring.brakeCompleted,
                         PT := T#1ms);
   IF #statTonTimer[61].Q THEN
       "Unit1.Em6.ControlNodes".cm.brakeTest.visionUnit.monitoring."step" := 20;
   END_IF;
   #_w2 := "Unit1.Em6.ControlNodes".cm.brakeTest.visionUnit.monitoring."step" = 20;
   IF #_w2 THEN "Unit1.Em6.ControlNodes".cm.brakeTest.visionUnit.commands.axisReset := TRUE; END_IF;
   #statTonTimer[62].TON(IN := #_w2 AND ("Unit1.Em6.ControlNodes".cmVisionUnitAxisZ.monitoring.resetActive OR "Unit1.Em6.ControlNodes".cmVisionUnitAxisZ.monitoring.axisEnabled),
                         PT := T#1ms);
   IF #statTonTimer[62].Q THEN
       "Unit1.Em6.ControlNodes".cm.brakeTest.visionUnit.monitoring."step" := 30;
   END_IF;
   #_w3 := "Unit1.Em6.ControlNodes".cm.brakeTest.visionUnit.monitoring."step" = 30;
   IF #_w3 THEN
       "Unit1.Em6.ControlNodes".cm.brakeTest.visionUnit.monitoring.busy := FALSE;
       "Unit1.Em6.ControlNodes".cm.brakeTest.visionUnit.commands.axisReset := FALSE;
       "Unit1.Em6.ControlNodes".cm.brakeTest.visionUnit.monitoring.complete := TRUE;
       "Unit1.Em6.ControlNodes".cmVisionUnitAxisZ.commands.enableAxis := FALSE;
       "Unit1.Em6.HmiInterface".cmVisionUnitAxisZ.commands.enableAxis := TRUE;
   END_IF;
   #statTonTimer[63].TON(IN := #_w3, PT := T#1ms);
   IF #statTonTimer[63].Q THEN
       "Unit1.Em6.ControlNodes".cm.brakeTest.visionUnit.monitoring."step" := 0;
   END_IF;
   #_w4 := "Unit1.EmNodes".devicesSummary.allDoorsOK AND NOT #statPulse[18];   // rising edge
   #statPulse[18] := "Unit1.EmNodes".devicesSummary.allDoorsOK;
   IF #_w4 THEN "Unit1.Em6.ControlNodes".cm.brakeTest.visionUnit.monitoring.complete := FALSE; END_IF;
END_REGION

REGION Network 66: Vision Z-Axis Brake Test Monitoring
   RUNG wire#powerrail
      Move(in := "Unit1.Em6.ControlNodes".cm.brakeTest.visionUnit.monitoring, out1 => "Unit1.Em6.HmiInterface".cm.brakeTest.visionUnit.monitoring)
   END_RUNG
   // the same network as SCL:
   "Unit1.Em6.HmiInterface".cm.brakeTest.visionUnit.monitoring := "Unit1.Em6.ControlNodes".cm.brakeTest.visionUnit.monitoring;
END_REGION

REGION Network 67: Call Vision Z-Axis Telegram 701
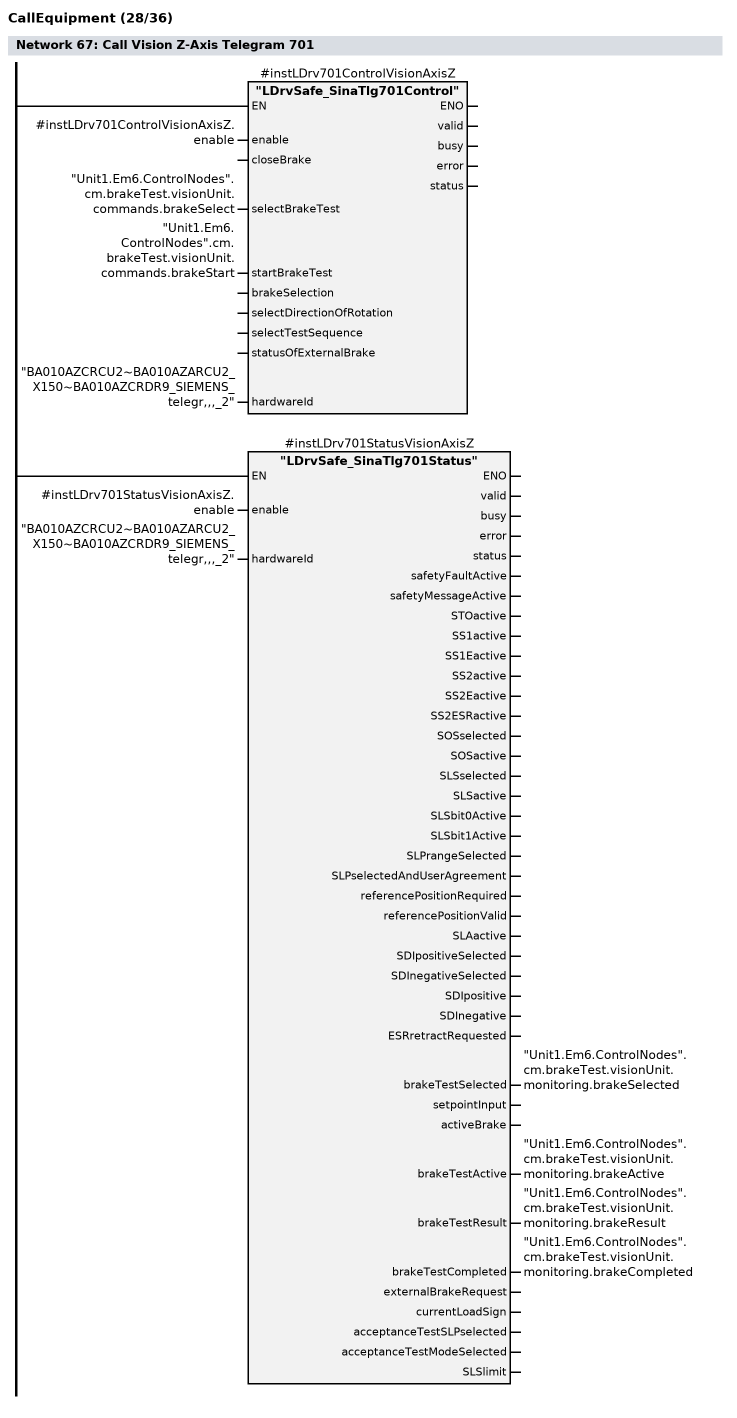
   RUNG wire#powerrail
      #instLDrv701ControlVisionAxisZ(enable := #instLDrv701ControlVisionAxisZ.enable, closeBrake :=, selectBrakeTest := "Unit1.Em6.ControlNodes".cm.brakeTest.visionUnit.commands.brakeSelect, startBrakeTest := "Unit1.Em6.ControlNodes".cm.brakeTest.visionUnit.commands.brakeStart, brakeSelection :=, selectDirectionOfRotation :=, selectTestSequence :=, statusOfExternalBrake :=, hardwareId := "BA010AZCRCU2~BA010AZARCU2_X150~BA010AZCRDR9_SIEMENS_telegr,,,_2", valid =>, busy =>, error =>, status =>)
   END_RUNG
   RUNG wire#powerrail
      #instLDrv701StatusVisionAxisZ(enable := #instLDrv701StatusVisionAxisZ.enable, hardwareId := "BA010AZCRCU2~BA010AZARCU2_X150~BA010AZCRDR9_SIEMENS_telegr,,,_2", valid =>, busy =>, error =>, status =>, safetyFaultActive =>, safetyMessageActive =>, STOactive =>, SS1active =>, SS1Eactive =>, SS2active =>, SS2Eactive =>, SS2ESRactive =>, SOSselected =>, SOSactive =>, SLSselected =>, SLSactive =>, SLSbit0Active =>, SLSbit1Active =>, SLPrangeSelected =>, SLPselectedAndUserAgreement =>, referencePositionRequired =>, referencePositionValid =>, SLAactive =>, SDIpositiveSelected =>, SDInegativeSelected =>, SDIpositive =>, SDInegative =>, ESRretractRequested =>, brakeTestSelected => "Unit1.Em6.ControlNodes".cm.brakeTest.visionUnit.monitoring.brakeSelected, setpointInput =>, activeBrake =>, brakeTestActive => "Unit1.Em6.ControlNodes".cm.brakeTest.visionUnit.monitoring.brakeActive, brakeTestResult => "Unit1.Em6.ControlNodes".cm.brakeTest.visionUnit.monitoring.brakeResult, brakeTestCompleted => "Unit1.Em6.ControlNodes".cm.brakeTest.visionUnit.monitoring.brakeCompleted, externalBrakeRequest =>, currentLoadSign =>, acceptanceTestSLPselected =>, acceptanceTestModeSelected =>, SLSlimit =>)
   END_RUNG
   // the same network as SCL:
   #instLDrv701ControlVisionAxisZ(enable := #instLDrv701ControlVisionAxisZ.enable,   // "LDrvSafe_SinaTlg701Control"
                           selectBrakeTest := "Unit1.Em6.ControlNodes".cm.brakeTest.visionUnit.commands.brakeSelect,
                           startBrakeTest := "Unit1.Em6.ControlNodes".cm.brakeTest.visionUnit.commands.brakeStart,
                           hardwareId := "BA010AZCRCU2~BA010AZARCU2_X150~BA010AZCRDR9_SIEMENS_telegr,,,_2");
   #instLDrv701StatusVisionAxisZ(enable := #instLDrv701StatusVisionAxisZ.enable,   // "LDrvSafe_SinaTlg701Status"
                           hardwareId := "BA010AZCRCU2~BA010AZARCU2_X150~BA010AZCRDR9_SIEMENS_telegr,,,_2",
                           brakeTestSelected => "Unit1.Em6.ControlNodes".cm.brakeTest.visionUnit.monitoring.brakeSelected,
                           brakeTestActive => "Unit1.Em6.ControlNodes".cm.brakeTest.visionUnit.monitoring.brakeActive,
                           brakeTestResult => "Unit1.Em6.ControlNodes".cm.brakeTest.visionUnit.monitoring.brakeResult,
                           brakeTestCompleted => "Unit1.Em6.ControlNodes".cm.brakeTest.visionUnit.monitoring.brakeCompleted);
END_REGION

REGION Network 69: ******************** Control Modules (TwoWayActuator) ********************
   // Call control modules that are actuators after the em logic (jobs and sequence), so that the latest commands are applied to the actuators.
END_REGION

REGION Network 70: Reset CMS
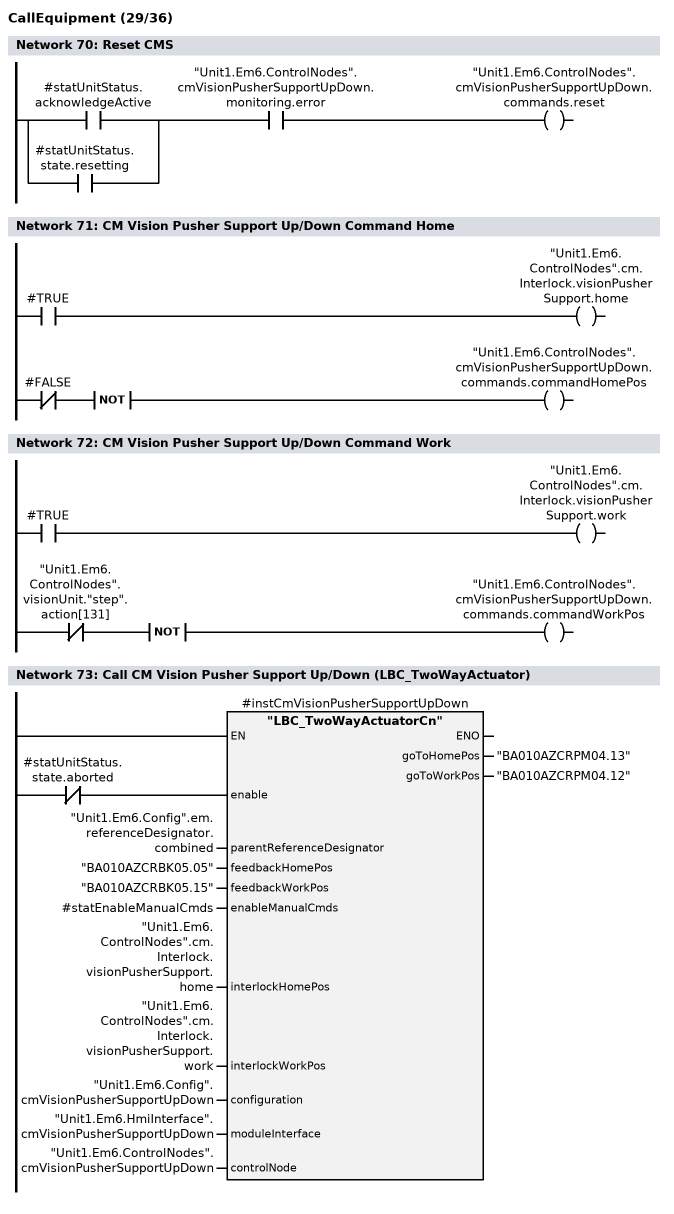
   RUNG wire#powerrail
      Contact( #statUnitStatus.acknowledgeActive )
      wire#w1
      Contact( "Unit1.Em6.ControlNodes".cmVisionPusherSupportUpDown.monitoring.error )
      Coil( "Unit1.Em6.ControlNodes".cmVisionPusherSupportUpDown.commands.reset )
   END_RUNG
   RUNG wire#powerrail
      Contact( #statUnitStatus.state.resetting )
   END_RUNG wire#w1
   // the same network as SCL:
   "Unit1.Em6.ControlNodes".cmVisionPusherSupportUpDown.commands.reset := (#statUnitStatus.acknowledgeActive OR #statUnitStatus.state.resetting) AND "Unit1.Em6.ControlNodes".cmVisionPusherSupportUpDown.monitoring.error;
END_REGION

REGION Network 71: CM Vision Pusher Support Up/Down Command Home
   RUNG wire#powerrail
      Contact( #TRUE )
      Coil( "Unit1.Em6.ControlNodes".cm.Interlock.visionPusherSupport.home )
   END_RUNG
   RUNG wire#powerrail
      I_Contact( #FALSE )
      Not()
      Coil( "Unit1.Em6.ControlNodes".cmVisionPusherSupportUpDown.commands.commandHomePos )
   END_RUNG
   // the same network as SCL:
   "Unit1.Em6.ControlNodes".cm.Interlock.visionPusherSupport.home := #TRUE;
   "Unit1.Em6.ControlNodes".cmVisionPusherSupportUpDown.commands.commandHomePos := NOT (NOT #FALSE);
END_REGION

REGION Network 72: CM Vision Pusher Support Up/Down Command Work
   RUNG wire#powerrail
      Contact( #TRUE )
      Coil( "Unit1.Em6.ControlNodes".cm.Interlock.visionPusherSupport.work )
   END_RUNG
   RUNG wire#powerrail
      I_Contact( "Unit1.Em6.ControlNodes".visionUnit."step".action[131] )
      Not()
      Coil( "Unit1.Em6.ControlNodes".cmVisionPusherSupportUpDown.commands.commandWorkPos )
   END_RUNG
   // the same network as SCL:
   "Unit1.Em6.ControlNodes".cm.Interlock.visionPusherSupport.work := #TRUE;
   "Unit1.Em6.ControlNodes".cmVisionPusherSupportUpDown.commands.commandWorkPos := NOT (NOT "Unit1.Em6.ControlNodes".visionUnit."step".action[131]);
END_REGION

REGION Network 73: Call CM Vision Pusher Support Up/Down (LBC_TwoWayActuator)
   RUNG wire#powerrail
      #instCmVisionPusherSupportUpDown(enable := wire#w1, parentReferenceDesignator := "Unit1.Em6.Config".em.referenceDesignator.combined, feedbackHomePos := "BA010AZCRBK05.05", feedbackWorkPos := "BA010AZCRBK05.15", enableManualCmds := #statEnableManualCmds, interlockHomePos := "Unit1.Em6.ControlNodes".cm.Interlock.visionPusherSupport.home, interlockWorkPos := "Unit1.Em6.ControlNodes".cm.Interlock.visionPusherSupport.work, configuration := "Unit1.Em6.Config".cmVisionPusherSupportUpDown, moduleInterface := "Unit1.Em6.HmiInterface".cmVisionPusherSupportUpDown, controlNode := "Unit1.Em6.ControlNodes".cmVisionPusherSupportUpDown, goToHomePos => "BA010AZCRPM04.13", goToWorkPos => "BA010AZCRPM04.12")
   END_RUNG
   RUNG wire#powerrail
      I_Contact( #statUnitStatus.state.aborted )
   END_RUNG wire#w1
   // the same network as SCL:
   #instCmVisionPusherSupportUpDown(enable := NOT #statUnitStatus.state.aborted,   // "LBC_TwoWayActuatorCn"
                           parentReferenceDesignator := "Unit1.Em6.Config".em.referenceDesignator.combined,
                           feedbackHomePos := "BA010AZCRBK05.05",
                           feedbackWorkPos := "BA010AZCRBK05.15",
                           enableManualCmds := #statEnableManualCmds,
                           interlockHomePos := "Unit1.Em6.ControlNodes".cm.Interlock.visionPusherSupport.home,
                           interlockWorkPos := "Unit1.Em6.ControlNodes".cm.Interlock.visionPusherSupport.work,
                           configuration := "Unit1.Em6.Config".cmVisionPusherSupportUpDown,
                           moduleInterface := "Unit1.Em6.HmiInterface".cmVisionPusherSupportUpDown,
                           controlNode := "Unit1.Em6.ControlNodes".cmVisionPusherSupportUpDown,
                           goToHomePos => "BA010AZCRPM04.13",
                           goToWorkPos => "BA010AZCRPM04.12");
END_REGION

REGION Network 74: ******************** Control Modules (Accessories) ********************
   // Call control modules that are actuators after the em logic (jobs and sequence), so that the latest commands are applied to the actuators.
END_REGION

REGION Network 75: Reset CMS
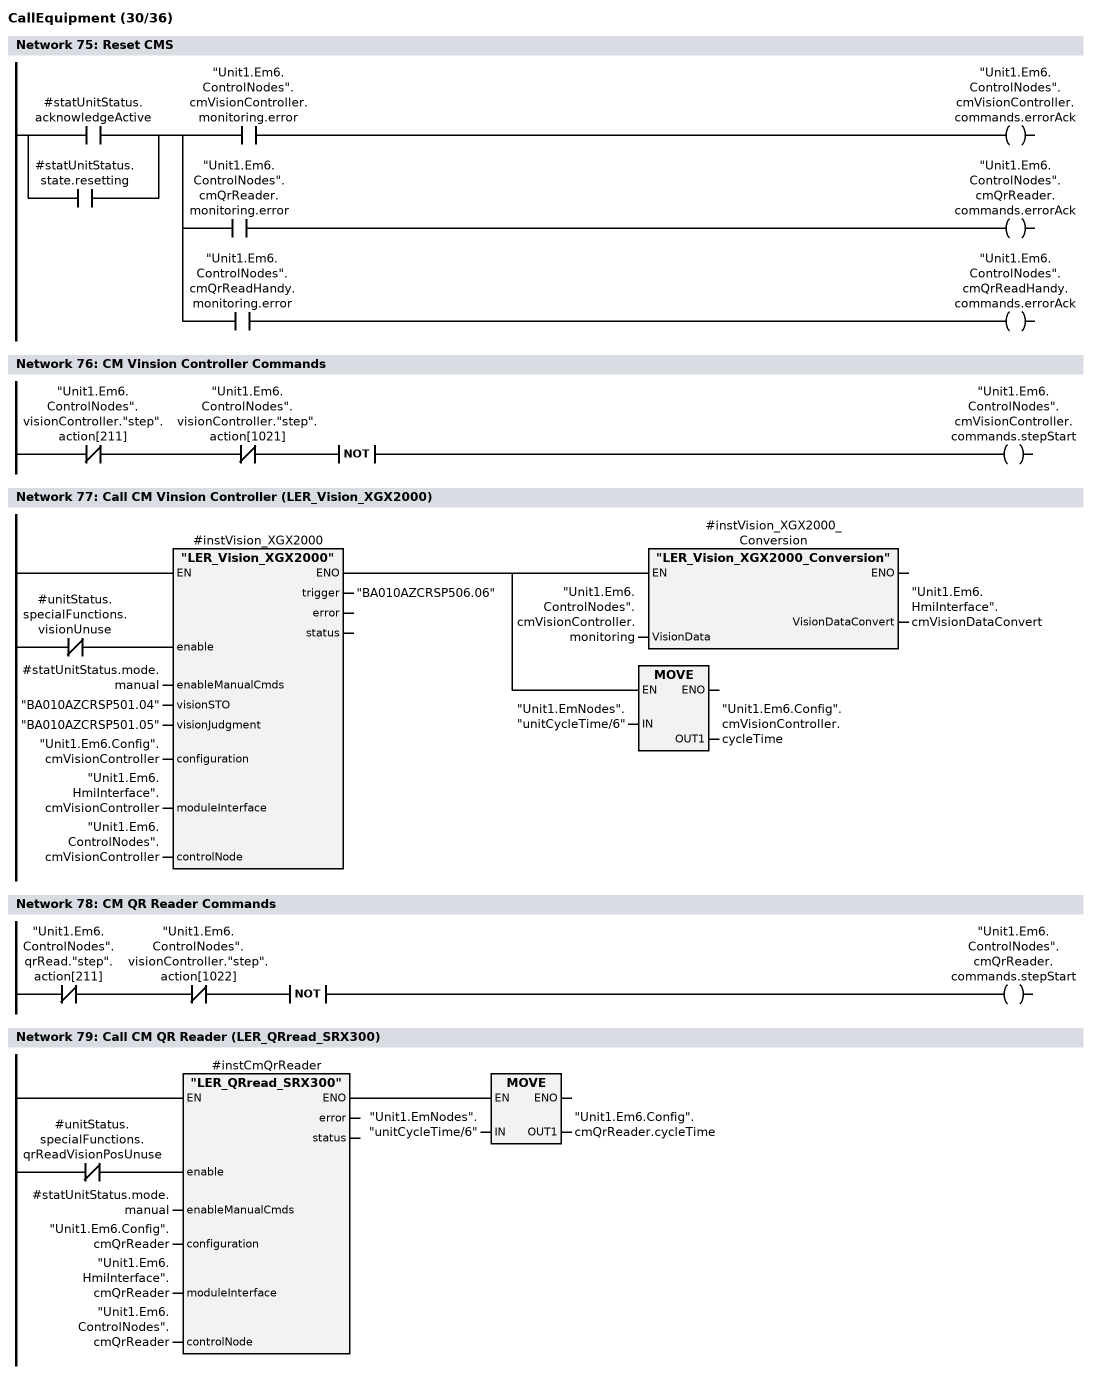
   RUNG wire#powerrail
      Contact( #statUnitStatus.acknowledgeActive )
      wire#w1
      Contact( "Unit1.Em6.ControlNodes".cmVisionController.monitoring.error )
      Coil( "Unit1.Em6.ControlNodes".cmVisionController.commands.errorAck )
   END_RUNG
   RUNG wire#powerrail
      Contact( #statUnitStatus.state.resetting )
   END_RUNG wire#w1
   RUNG wire#w1
      Contact( "Unit1.Em6.ControlNodes".cmQrReader.monitoring.error )
      Coil( "Unit1.Em6.ControlNodes".cmQrReader.commands.errorAck )
   END_RUNG
   RUNG wire#w1
      Contact( "Unit1.Em6.ControlNodes".cmQrReadHandy.monitoring.error )
      Coil( "Unit1.Em6.ControlNodes".cmQrReadHandy.commands.errorAck )
   END_RUNG
   // the same network as SCL:
   #_w1 := #statUnitStatus.acknowledgeActive OR #statUnitStatus.state.resetting;
   "Unit1.Em6.ControlNodes".cmVisionController.commands.errorAck := #_w1 AND "Unit1.Em6.ControlNodes".cmVisionController.monitoring.error;
   "Unit1.Em6.ControlNodes".cmQrReader.commands.errorAck := #_w1 AND "Unit1.Em6.ControlNodes".cmQrReader.monitoring.error;
   "Unit1.Em6.ControlNodes".cmQrReadHandy.commands.errorAck := #_w1 AND "Unit1.Em6.ControlNodes".cmQrReadHandy.monitoring.error;
END_REGION

REGION Network 76: CM Vinsion Controller Commands
   RUNG wire#powerrail
      I_Contact( "Unit1.Em6.ControlNodes".visionController."step".action[211] )
      I_Contact( "Unit1.Em6.ControlNodes".visionController."step".action[1021] )
      Not()
      Coil( "Unit1.Em6.ControlNodes".cmVisionController.commands.stepStart )
   END_RUNG
   // the same network as SCL:
   "Unit1.Em6.ControlNodes".cmVisionController.commands.stepStart := NOT (NOT "Unit1.Em6.ControlNodes".visionController."step".action[211] AND NOT "Unit1.Em6.ControlNodes".visionController."step".action[1021]);
END_REGION

REGION Network 77: Call CM Vinsion Controller (LER_Vision_XGX2000)
   RUNG wire#powerrail
      #instVision_XGX2000(enable := wire#w1, enableManualCmds := #statUnitStatus.mode.manual, visionSTO := "BA010AZCRSP501.04", visionJudgment := "BA010AZCRSP501.05", configuration := "Unit1.Em6.Config".cmVisionController, moduleInterface := "Unit1.Em6.HmiInterface".cmVisionController, controlNode := "Unit1.Em6.ControlNodes".cmVisionController, trigger => "BA010AZCRSP506.06", error =>, status =>)
      wire#w2
      #instVision_XGX2000_Conversion(VisionData := "Unit1.Em6.ControlNodes".cmVisionController.monitoring, VisionDataConvert => "Unit1.Em6.HmiInterface".cmVisionDataConvert)
   END_RUNG
   RUNG wire#powerrail
      I_Contact( #unitStatus.specialFunctions.visionUnuse )
   END_RUNG wire#w1
   RUNG wire#w2
      Move(in := "Unit1.EmNodes"."unitCycleTime/6", out1 => "Unit1.Em6.Config".cmVisionController.cycleTime)
   END_RUNG
   // the same network as SCL:
   #instVision_XGX2000(enable := NOT #unitStatus.specialFunctions.visionUnuse,   // "LER_Vision_XGX2000"
                       enableManualCmds := #statUnitStatus.mode.manual,
                       visionSTO := "BA010AZCRSP501.04",
                       visionJudgment := "BA010AZCRSP501.05",
                       configuration := "Unit1.Em6.Config".cmVisionController,
                       moduleInterface := "Unit1.Em6.HmiInterface".cmVisionController,
                       controlNode := "Unit1.Em6.ControlNodes".cmVisionController,
                       trigger => "BA010AZCRSP506.06",
                       ENO => #_w1);
   IF #_w1 THEN
       #instVision_XGX2000_Conversion(VisionData := "Unit1.Em6.ControlNodes".cmVisionController.monitoring,   // "LER_Vision_XGX2000_Conversion"
                               VisionDataConvert => "Unit1.Em6.HmiInterface".cmVisionDataConvert);
       "Unit1.Em6.Config".cmVisionController.cycleTime := "Unit1.EmNodes"."unitCycleTime/6";
   END_IF;
END_REGION

REGION Network 78: CM QR Reader Commands
   RUNG wire#powerrail
      I_Contact( "Unit1.Em6.ControlNodes".qrRead."step".action[211] )
      I_Contact( "Unit1.Em6.ControlNodes".visionController."step".action[1022] )
      Not()
      Coil( "Unit1.Em6.ControlNodes".cmQrReader.commands.stepStart )
   END_RUNG
   // the same network as SCL:
   "Unit1.Em6.ControlNodes".cmQrReader.commands.stepStart := NOT (NOT "Unit1.Em6.ControlNodes".qrRead."step".action[211] AND NOT "Unit1.Em6.ControlNodes".visionController."step".action[1022]);
END_REGION

REGION Network 79: Call CM QR Reader (LER_QRread_SRX300)
   RUNG wire#powerrail
      #instCmQrReader(enable := wire#w1, enableManualCmds := #statUnitStatus.mode.manual, configuration := "Unit1.Em6.Config".cmQrReader, moduleInterface := "Unit1.Em6.HmiInterface".cmQrReader, controlNode := "Unit1.Em6.ControlNodes".cmQrReader, error =>, status =>)
      Move(in := "Unit1.EmNodes"."unitCycleTime/6", out1 => "Unit1.Em6.Config".cmQrReader.cycleTime)
   END_RUNG
   RUNG wire#powerrail
      I_Contact( #unitStatus.specialFunctions.qrReadVisionPosUnuse )
   END_RUNG wire#w1
   // the same network as SCL:
   #instCmQrReader(enable := NOT #unitStatus.specialFunctions.qrReadVisionPosUnuse,   // "LER_QRread_SRX300"
                   enableManualCmds := #statUnitStatus.mode.manual,
                   configuration := "Unit1.Em6.Config".cmQrReader,
                   moduleInterface := "Unit1.Em6.HmiInterface".cmQrReader,
                   controlNode := "Unit1.Em6.ControlNodes".cmQrReader,
                   ENO => #_w1);
   IF #_w1 THEN "Unit1.Em6.Config".cmQrReader.cycleTime := "Unit1.EmNodes"."unitCycleTime/6"; END_IF;
END_REGION

REGION Network 80: Call CM QR Reader Handy (LER_QRread_DM8700)
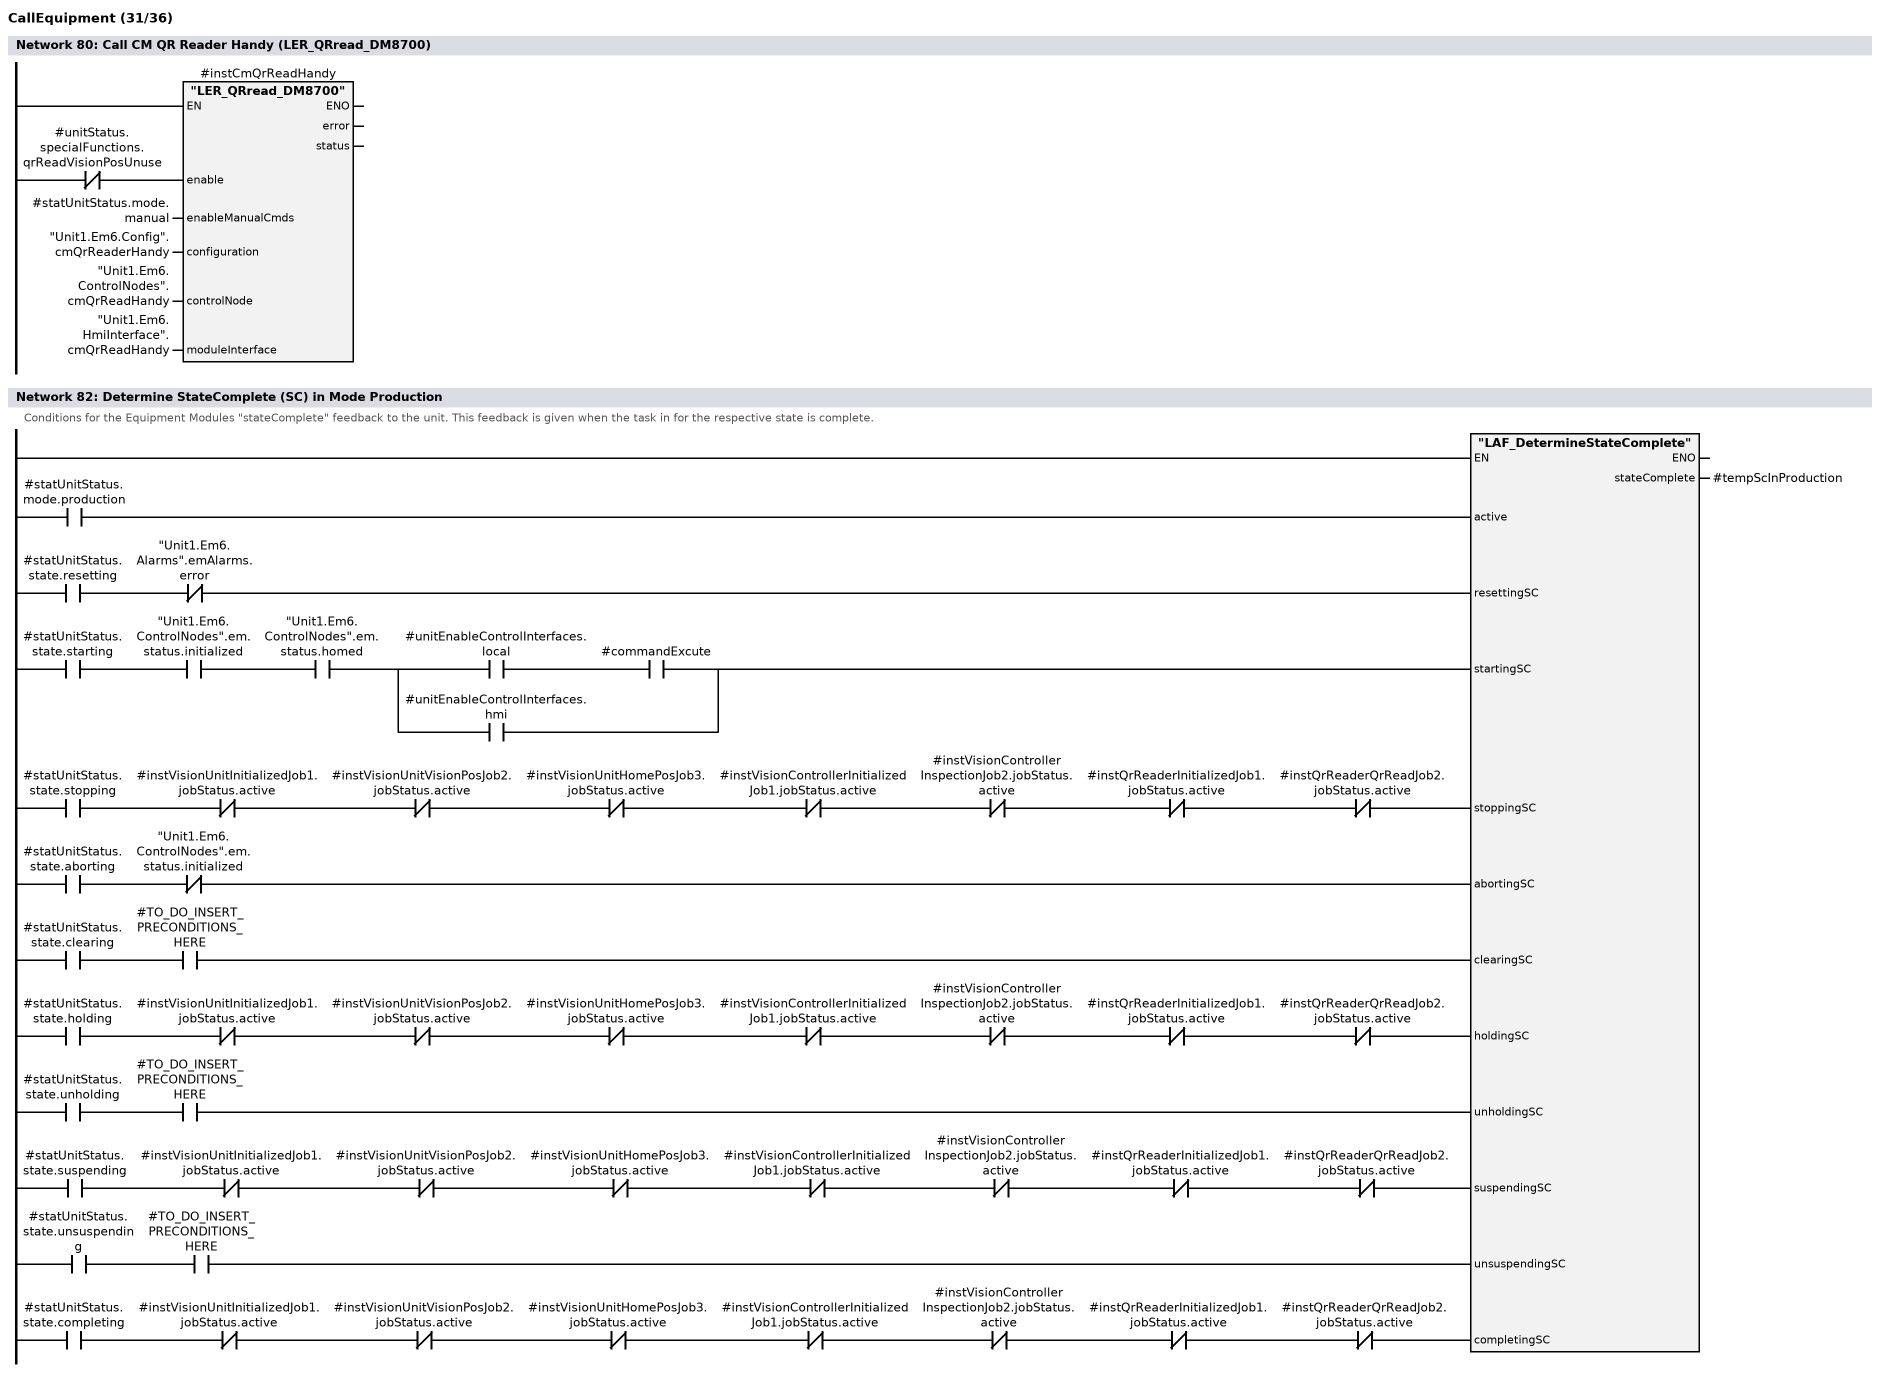
   RUNG wire#powerrail
      #instCmQrReadHandy(enable := wire#w1, enableManualCmds := #statUnitStatus.mode.manual, configuration := "Unit1.Em6.Config".cmQrReaderHandy, controlNode := "Unit1.Em6.ControlNodes".cmQrReadHandy, moduleInterface := "Unit1.Em6.HmiInterface".cmQrReadHandy, error =>, status =>)
   END_RUNG
   RUNG wire#powerrail
      I_Contact( #unitStatus.specialFunctions.qrReadVisionPosUnuse )
   END_RUNG wire#w1
   // the same network as SCL:
   #instCmQrReadHandy(enable := NOT #unitStatus.specialFunctions.qrReadVisionPosUnuse,   // "LER_QRread_DM8700"
                      enableManualCmds := #statUnitStatus.mode.manual,
                      configuration := "Unit1.Em6.Config".cmQrReaderHandy,
                      controlNode := "Unit1.Em6.ControlNodes".cmQrReadHandy,
                      moduleInterface := "Unit1.Em6.HmiInterface".cmQrReadHandy);
END_REGION

REGION Network 81: ******************** Feedback to Unit ********************
END_REGION

REGION Network 82: Determine StateComplete (SC) in Mode Production
   // Conditions for the Equipment Modules "stateComplete" feedback to the unit. This feedback is given when the task in for the respective state is complete.
   RUNG wire#powerrail
      "LAF_DetermineStateComplete"(active := wire#w1, resettingSC := wire#w2, startingSC := wire#w4, stoppingSC := wire#w5, abortingSC := wire#w6, clearingSC := wire#w7, holdingSC := wire#w8, unholdingSC := wire#w9, suspendingSC := wire#w10, unsuspendingSC := wire#w11, completingSC := wire#w12, stateComplete => #tempScInProduction)
   END_RUNG
   RUNG wire#powerrail
      Contact( #statUnitStatus.mode.production )
   END_RUNG wire#w1
   RUNG wire#powerrail
      Contact( #statUnitStatus.state.resetting )
      I_Contact( "Unit1.Em6.Alarms".emAlarms.error )
   END_RUNG wire#w2
   RUNG wire#powerrail
      Contact( #statUnitStatus.state.starting )
      Contact( "Unit1.Em6.ControlNodes".em.status.initialized )
      Contact( "Unit1.Em6.ControlNodes".em.status.homed )
      wire#w3
      Contact( #unitEnableControlInterfaces.local )
      Contact( #commandExcute )
   END_RUNG wire#w4
   RUNG wire#w3
      Contact( #unitEnableControlInterfaces.hmi )
   END_RUNG wire#w4
   RUNG wire#powerrail
      Contact( #statUnitStatus.state.stopping )
      I_Contact( #instVisionUnitInitializedJob1.jobStatus.active )
      I_Contact( #instVisionUnitVisionPosJob2.jobStatus.active )
      I_Contact( #instVisionUnitHomePosJob3.jobStatus.active )
      I_Contact( #instVisionControllerInitializedJob1.jobStatus.active )
      I_Contact( #instVisionControllerInspectionJob2.jobStatus.active )
      I_Contact( #instQrReaderInitializedJob1.jobStatus.active )
      I_Contact( #instQrReaderQrReadJob2.jobStatus.active )
   END_RUNG wire#w5
   RUNG wire#powerrail
      Contact( #statUnitStatus.state.aborting )
      I_Contact( "Unit1.Em6.ControlNodes".em.status.initialized )
   END_RUNG wire#w6
   RUNG wire#powerrail
      Contact( #statUnitStatus.state.clearing )
      Contact( #TO_DO_INSERT_PRECONDITIONS_HERE )
   END_RUNG wire#w7
   RUNG wire#powerrail
      Contact( #statUnitStatus.state.holding )
      I_Contact( #instVisionUnitInitializedJob1.jobStatus.active )
      I_Contact( #instVisionUnitVisionPosJob2.jobStatus.active )
      I_Contact( #instVisionUnitHomePosJob3.jobStatus.active )
      I_Contact( #instVisionControllerInitializedJob1.jobStatus.active )
      I_Contact( #instVisionControllerInspectionJob2.jobStatus.active )
      I_Contact( #instQrReaderInitializedJob1.jobStatus.active )
      I_Contact( #instQrReaderQrReadJob2.jobStatus.active )
   END_RUNG wire#w8
   RUNG wire#powerrail
      Contact( #statUnitStatus.state.unholding )
      Contact( #TO_DO_INSERT_PRECONDITIONS_HERE )
   END_RUNG wire#w9
   RUNG wire#powerrail
      Contact( #statUnitStatus.state.suspending )
      I_Contact( #instVisionUnitInitializedJob1.jobStatus.active )
      I_Contact( #instVisionUnitVisionPosJob2.jobStatus.active )
      I_Contact( #instVisionUnitHomePosJob3.jobStatus.active )
      I_Contact( #instVisionControllerInitializedJob1.jobStatus.active )
      I_Contact( #instVisionControllerInspectionJob2.jobStatus.active )
      I_Contact( #instQrReaderInitializedJob1.jobStatus.active )
      I_Contact( #instQrReaderQrReadJob2.jobStatus.active )
   END_RUNG wire#w10
   RUNG wire#powerrail
      Contact( #statUnitStatus.state.unsuspending )
      Contact( #TO_DO_INSERT_PRECONDITIONS_HERE )
   END_RUNG wire#w11
   RUNG wire#powerrail
      Contact( #statUnitStatus.state.completing )
      I_Contact( #instVisionUnitInitializedJob1.jobStatus.active )
      I_Contact( #instVisionUnitVisionPosJob2.jobStatus.active )
      I_Contact( #instVisionUnitHomePosJob3.jobStatus.active )
      I_Contact( #instVisionControllerInitializedJob1.jobStatus.active )
      I_Contact( #instVisionControllerInspectionJob2.jobStatus.active )
      I_Contact( #instQrReaderInitializedJob1.jobStatus.active )
      I_Contact( #instQrReaderQrReadJob2.jobStatus.active )
   END_RUNG wire#w12
   // the same network as SCL:
   "LAF_DetermineStateComplete"(active := #statUnitStatus.mode.production,
                           resettingSC := #statUnitStatus.state.resetting AND NOT "Unit1.Em6.Alarms".emAlarms.error,
                           startingSC := #statUnitStatus.state.starting AND "Unit1.Em6.ControlNodes".em.status.initialized AND "Unit1.Em6.ControlNodes".em.status.homed AND ((#unitEnableControlInterfaces.local AND #commandExcute) OR #unitEnableControlInterfaces.hmi),
                           stoppingSC := #statUnitStatus.state.stopping AND NOT #instVisionUnitInitializedJob1.jobStatus.active AND NOT #instVisionUnitVisionPosJob2.jobStatus.active AND NOT #instVisionUnitHomePosJob3.jobStatus.active AND NOT #instVisionControllerInitializedJob1.jobStatus.active AND NOT #instVisionControllerInspectionJob2.jobStatus.active AND NOT #instQrReaderInitializedJob1.jobStatus.active AND NOT #instQrReaderQrReadJob2.jobStatus.active,
                           abortingSC := #statUnitStatus.state.aborting AND NOT "Unit1.Em6.ControlNodes".em.status.initialized,
                           clearingSC := #statUnitStatus.state.clearing AND #TO_DO_INSERT_PRECONDITIONS_HERE,
                           holdingSC := #statUnitStatus.state.holding AND NOT #instVisionUnitInitializedJob1.jobStatus.active AND NOT #instVisionUnitVisionPosJob2.jobStatus.active AND NOT #instVisionUnitHomePosJob3.jobStatus.active AND NOT #instVisionControllerInitializedJob1.jobStatus.active AND NOT #instVisionControllerInspectionJob2.jobStatus.active AND NOT #instQrReaderInitializedJob1.jobStatus.active AND NOT #instQrReaderQrReadJob2.jobStatus.active,
                           unholdingSC := #statUnitStatus.state.unholding AND #TO_DO_INSERT_PRECONDITIONS_HERE,
                           suspendingSC := #statUnitStatus.state.suspending AND NOT #instVisionUnitInitializedJob1.jobStatus.active AND NOT #instVisionUnitVisionPosJob2.jobStatus.active AND NOT #instVisionUnitHomePosJob3.jobStatus.active AND NOT #instVisionControllerInitializedJob1.jobStatus.active AND NOT #instVisionControllerInspectionJob2.jobStatus.active AND NOT #instQrReaderInitializedJob1.jobStatus.active AND NOT #instQrReaderQrReadJob2.jobStatus.active,
                           unsuspendingSC := #statUnitStatus.state.unsuspending AND #TO_DO_INSERT_PRECONDITIONS_HERE,
                           completingSC := #statUnitStatus.state.completing AND NOT #instVisionUnitInitializedJob1.jobStatus.active AND NOT #instVisionUnitVisionPosJob2.jobStatus.active AND NOT #instVisionUnitHomePosJob3.jobStatus.active AND NOT #instVisionControllerInitializedJob1.jobStatus.active AND NOT #instVisionControllerInspectionJob2.jobStatus.active AND NOT #instQrReaderInitializedJob1.jobStatus.active AND NOT #instQrReaderQrReadJob2.jobStatus.active,
                           stateComplete => #tempScInProduction);
END_REGION

REGION Network 83: Determine StateComplete (SC) in Mode Maintenance/Manual
   // Conditions for the Equipment Modules "stateComplete" feedback to the unit. This feedback is given when the task in for the respective state is complete.
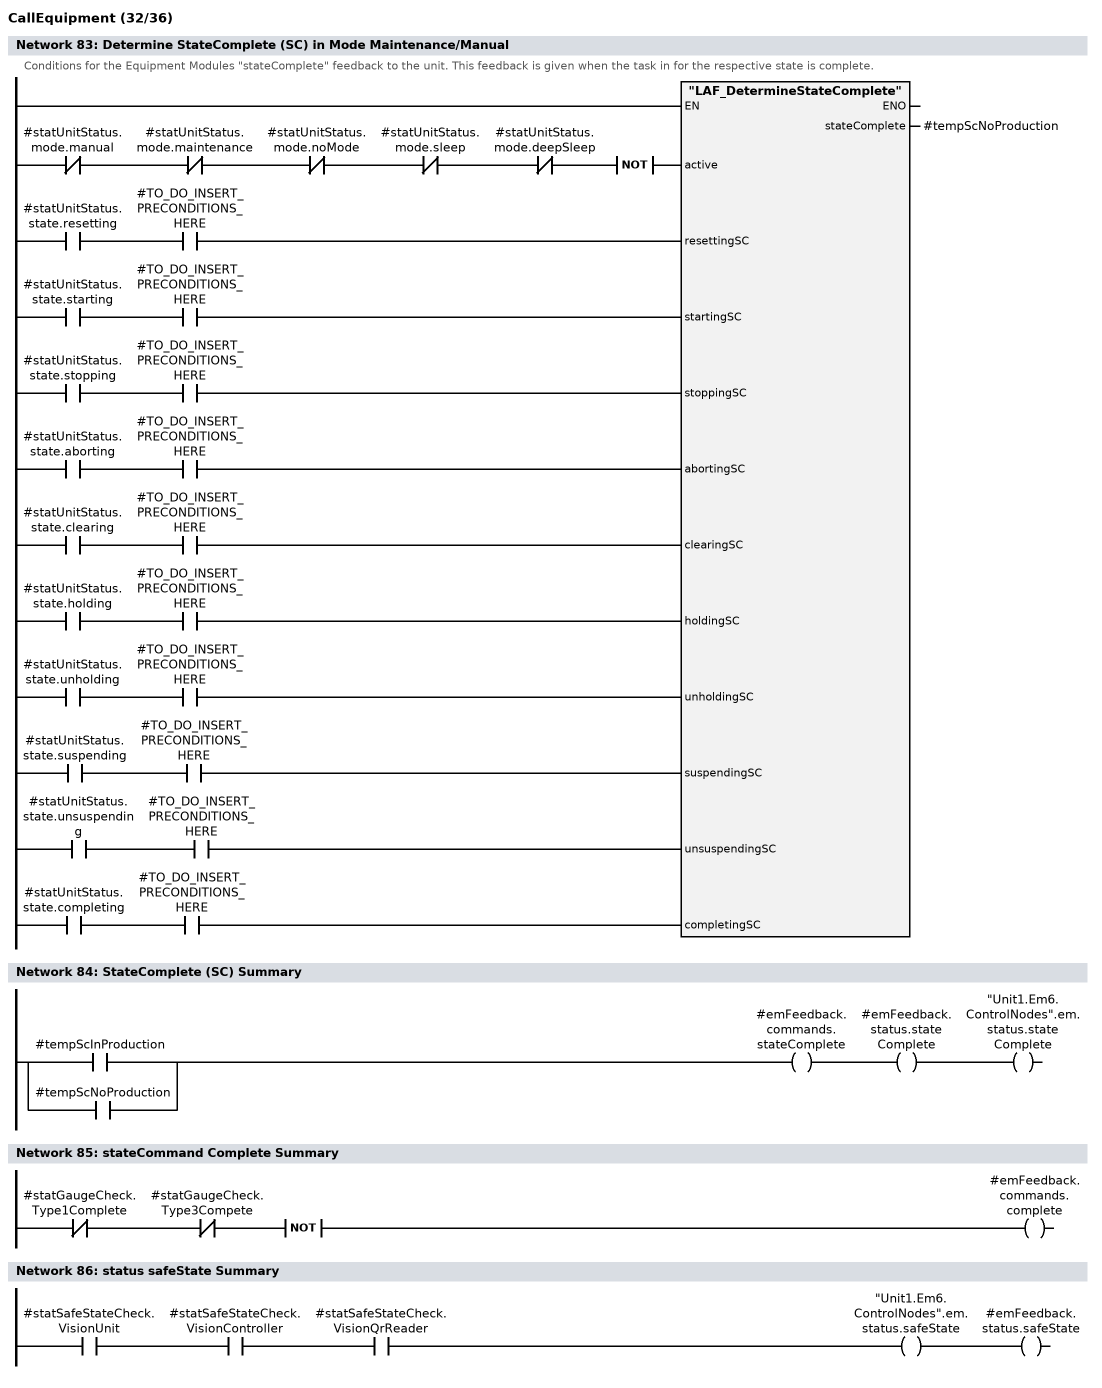
   RUNG wire#powerrail
      "LAF_DetermineStateComplete"(active := wire#w1, resettingSC := wire#w2, startingSC := wire#w3, stoppingSC := wire#w4, abortingSC := wire#w5, clearingSC := wire#w6, holdingSC := wire#w7, unholdingSC := wire#w8, suspendingSC := wire#w9, unsuspendingSC := wire#w10, completingSC := wire#w11, stateComplete => #tempScNoProduction)
   END_RUNG
   RUNG wire#powerrail
      I_Contact( #statUnitStatus.mode.manual )
      I_Contact( #statUnitStatus.mode.maintenance )
      I_Contact( #statUnitStatus.mode.noMode )
      I_Contact( #statUnitStatus.mode.sleep )
      I_Contact( #statUnitStatus.mode.deepSleep )
      Not()
   END_RUNG wire#w1
   RUNG wire#powerrail
      Contact( #statUnitStatus.state.resetting )
      Contact( #TO_DO_INSERT_PRECONDITIONS_HERE )
   END_RUNG wire#w2
   RUNG wire#powerrail
      Contact( #statUnitStatus.state.starting )
      Contact( #TO_DO_INSERT_PRECONDITIONS_HERE )
   END_RUNG wire#w3
   RUNG wire#powerrail
      Contact( #statUnitStatus.state.stopping )
      Contact( #TO_DO_INSERT_PRECONDITIONS_HERE )
   END_RUNG wire#w4
   RUNG wire#powerrail
      Contact( #statUnitStatus.state.aborting )
      Contact( #TO_DO_INSERT_PRECONDITIONS_HERE )
   END_RUNG wire#w5
   RUNG wire#powerrail
      Contact( #statUnitStatus.state.clearing )
      Contact( #TO_DO_INSERT_PRECONDITIONS_HERE )
   END_RUNG wire#w6
   RUNG wire#powerrail
      Contact( #statUnitStatus.state.holding )
      Contact( #TO_DO_INSERT_PRECONDITIONS_HERE )
   END_RUNG wire#w7
   RUNG wire#powerrail
      Contact( #statUnitStatus.state.unholding )
      Contact( #TO_DO_INSERT_PRECONDITIONS_HERE )
   END_RUNG wire#w8
   RUNG wire#powerrail
      Contact( #statUnitStatus.state.suspending )
      Contact( #TO_DO_INSERT_PRECONDITIONS_HERE )
   END_RUNG wire#w9
   RUNG wire#powerrail
      Contact( #statUnitStatus.state.unsuspending )
      Contact( #TO_DO_INSERT_PRECONDITIONS_HERE )
   END_RUNG wire#w10
   RUNG wire#powerrail
      Contact( #statUnitStatus.state.completing )
      Contact( #TO_DO_INSERT_PRECONDITIONS_HERE )
   END_RUNG wire#w11
   // the same network as SCL:
   "LAF_DetermineStateComplete"(active := NOT (NOT #statUnitStatus.mode.manual AND NOT #statUnitStatus.mode.maintenance AND NOT #statUnitStatus.mode.noMode AND NOT #statUnitStatus.mode.sleep AND NOT #statUnitStatus.mode.deepSleep),
                           resettingSC := #statUnitStatus.state.resetting AND #TO_DO_INSERT_PRECONDITIONS_HERE,
                           startingSC := #statUnitStatus.state.starting AND #TO_DO_INSERT_PRECONDITIONS_HERE,
                           stoppingSC := #statUnitStatus.state.stopping AND #TO_DO_INSERT_PRECONDITIONS_HERE,
                           abortingSC := #statUnitStatus.state.aborting AND #TO_DO_INSERT_PRECONDITIONS_HERE,
                           clearingSC := #statUnitStatus.state.clearing AND #TO_DO_INSERT_PRECONDITIONS_HERE,
                           holdingSC := #statUnitStatus.state.holding AND #TO_DO_INSERT_PRECONDITIONS_HERE,
                           unholdingSC := #statUnitStatus.state.unholding AND #TO_DO_INSERT_PRECONDITIONS_HERE,
                           suspendingSC := #statUnitStatus.state.suspending AND #TO_DO_INSERT_PRECONDITIONS_HERE,
                           unsuspendingSC := #statUnitStatus.state.unsuspending AND #TO_DO_INSERT_PRECONDITIONS_HERE,
                           completingSC := #statUnitStatus.state.completing AND #TO_DO_INSERT_PRECONDITIONS_HERE,
                           stateComplete => #tempScNoProduction);
END_REGION

REGION Network 84: StateComplete (SC) Summary
   RUNG wire#powerrail
      Contact( #tempScInProduction )
      wire#w1
      Coil( #emFeedback.commands.stateComplete )
      Coil( #emFeedback.status.stateComplete )
      Coil( "Unit1.Em6.ControlNodes".em.status.stateComplete )
   END_RUNG
   RUNG wire#powerrail
      Contact( #tempScNoProduction )
   END_RUNG wire#w1
   // the same network as SCL:
   #emFeedback.commands.stateComplete := #tempScInProduction OR #tempScNoProduction;
   #emFeedback.status.stateComplete := #emFeedback.commands.stateComplete;
   "Unit1.Em6.ControlNodes".em.status.stateComplete := #emFeedback.commands.stateComplete;
END_REGION

REGION Network 85: stateCommand Complete Summary
   RUNG wire#powerrail
      I_Contact( #statGaugeCheck.Type1Complete )
      I_Contact( #statGaugeCheck.Type3Compete )
      Not()
      Coil( #emFeedback.commands.complete )
   END_RUNG
   // the same network as SCL:
   #emFeedback.commands.complete := NOT (NOT #statGaugeCheck.Type1Complete AND NOT #statGaugeCheck.Type3Compete);
END_REGION

REGION Network 86: status safeState Summary
   RUNG wire#powerrail
      Contact( #statSafeStateCheck.VisionUnit )
      Contact( #statSafeStateCheck.VisionController )
      Contact( #statSafeStateCheck.VisionQrReader )
      Coil( "Unit1.Em6.ControlNodes".em.status.safeState )
      Coil( #emFeedback.status.safeState )
   END_RUNG
   // the same network as SCL:
   "Unit1.Em6.ControlNodes".em.status.safeState := #statSafeStateCheck.VisionUnit AND #statSafeStateCheck.VisionController AND #statSafeStateCheck.VisionQrReader;
   #emFeedback.status.safeState := "Unit1.Em6.ControlNodes".em.status.safeState;
END_REGION

REGION Network 87: status safetyReleased Summary
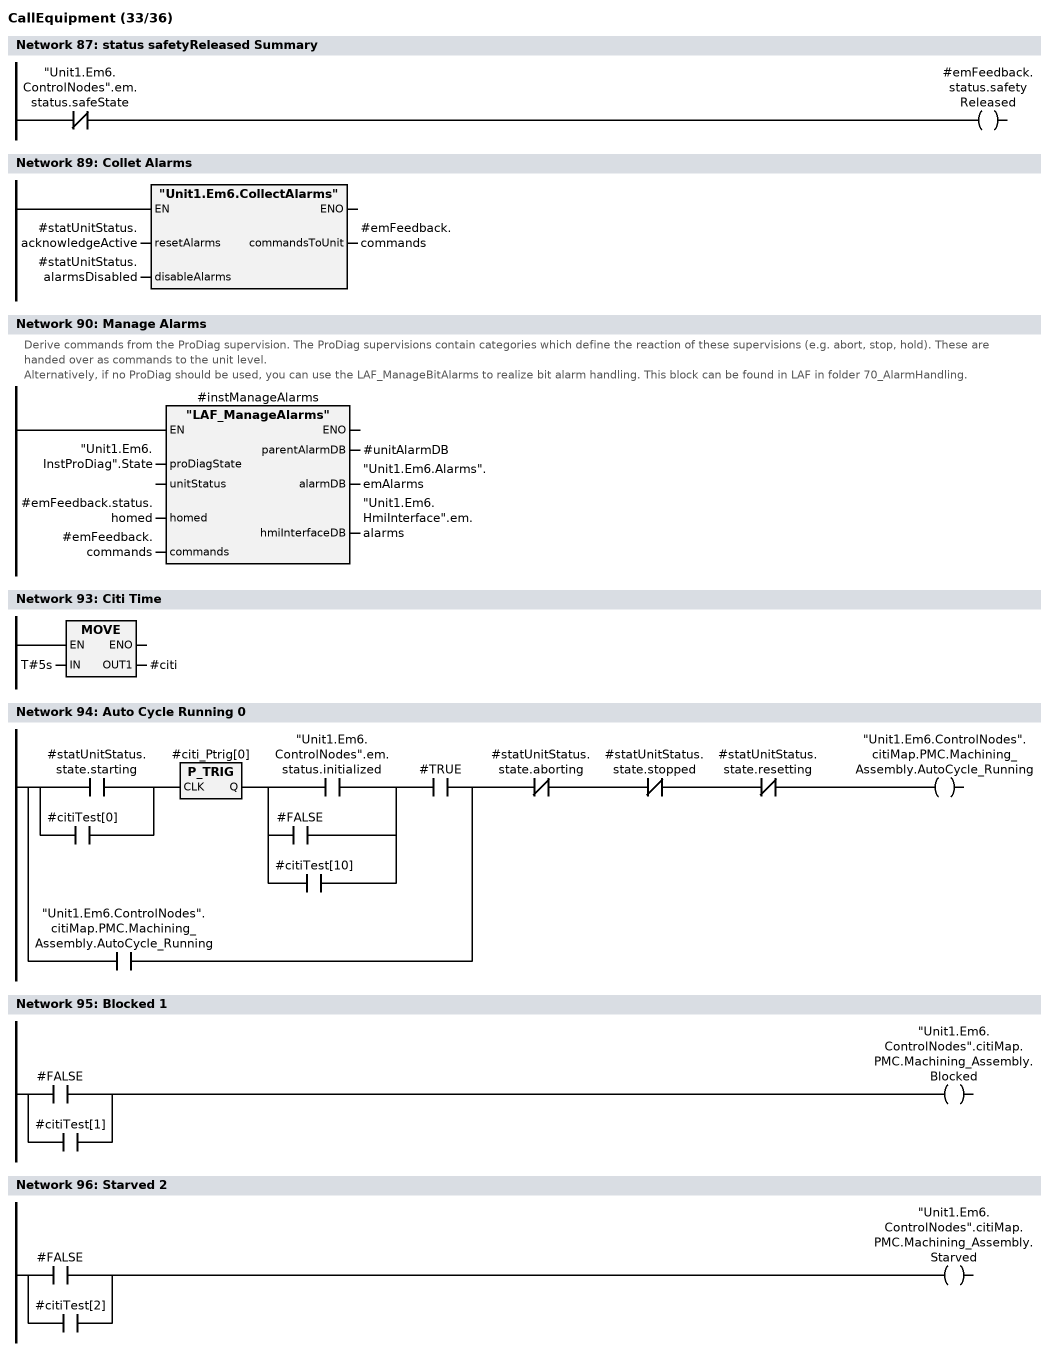
   RUNG wire#powerrail
      I_Contact( "Unit1.Em6.ControlNodes".em.status.safeState )
      Coil( #emFeedback.status.safetyReleased )
   END_RUNG
   // the same network as SCL:
   #emFeedback.status.safetyReleased := NOT "Unit1.Em6.ControlNodes".em.status.safeState;
END_REGION

REGION Network 88: ******************** Alarms ********************
END_REGION

REGION Network 89: Collet Alarms
   RUNG wire#powerrail
      "Unit1.Em6.CollectAlarms"(resetAlarms := #statUnitStatus.acknowledgeActive, disableAlarms := #statUnitStatus.alarmsDisabled, commandsToUnit => #emFeedback.commands)
   END_RUNG
   // the same network as SCL:
   "Unit1.Em6.CollectAlarms"(resetAlarms := #statUnitStatus.acknowledgeActive,
                           disableAlarms := #statUnitStatus.alarmsDisabled,
                           commandsToUnit => #emFeedback.commands);
END_REGION

REGION Network 90: Manage Alarms
   // Derive commands from the ProDiag supervision. The ProDiag supervisions contain categories which define the reaction of these supervisions (e.g. abort, stop, hold). These are handed over as commands to the unit level.
   // Alternatively, if no ProDiag should be used, you can use the LAF_ManageBitAlarms to realize bit alarm handling. This block can be found in LAF in folder 70_AlarmHandling.
   RUNG wire#powerrail
      #instManageAlarms(proDiagState := "Unit1.Em6.InstProDiag".State, unitStatus :=, homed := #emFeedback.status.homed, commands := #emFeedback.commands, parentAlarmDB => #unitAlarmDB, alarmDB => "Unit1.Em6.Alarms".emAlarms, hmiInterfaceDB => "Unit1.Em6.HmiInterface".em.alarms)
   END_RUNG
   // the same network as SCL:
   #instManageAlarms(proDiagState := "Unit1.Em6.InstProDiag".State,   // "LAF_ManageAlarms"
                     homed := #emFeedback.status.homed,
                     commands := #emFeedback.commands,
                     parentAlarmDB => #unitAlarmDB,
                     alarmDB => "Unit1.Em6.Alarms".emAlarms,
                     hmiInterfaceDB => "Unit1.Em6.HmiInterface".em.alarms);
END_REGION

REGION Network 92: ******************** CITI ********************
END_REGION

REGION Network 93: Citi Time
   RUNG wire#powerrail
      Move(in := T#5s, out1 => #citi)
   END_RUNG
   // the same network as SCL:
   #citi := T#5s;
END_REGION

REGION Network 94: Auto Cycle Running 0
   RUNG wire#powerrail
      Contact( #statUnitStatus.state.starting )
      wire#w1
      P_Trig( #citi_Ptrig[0] )
      wire#w2
      Contact( "Unit1.Em6.ControlNodes".em.status.initialized )
      wire#w3
      Contact( #TRUE )
      wire#w4
      I_Contact( #statUnitStatus.state.aborting )
      I_Contact( #statUnitStatus.state.stopped )
      I_Contact( #statUnitStatus.state.resetting )
      Coil( "Unit1.Em6.ControlNodes".citiMap.PMC.Machining_Assembly.AutoCycle_Running )
   END_RUNG
   RUNG wire#powerrail
      Contact( #citiTest[0] )
   END_RUNG wire#w1
   RUNG wire#w2
      Contact( #FALSE )
   END_RUNG wire#w3
   RUNG wire#w2
      Contact( #citiTest[10] )
   END_RUNG wire#w3
   RUNG wire#powerrail
      Contact( "Unit1.Em6.ControlNodes".citiMap.PMC.Machining_Assembly.AutoCycle_Running )
   END_RUNG wire#w4
   // the same network as SCL:
   #_w1 := #statUnitStatus.state.starting OR #citiTest[0];
   #_w2 := #_w1 AND NOT #citi_Ptrig[0];   // rising edge
   #citi_Ptrig[0] := #_w1;
   "Unit1.Em6.ControlNodes".citiMap.PMC.Machining_Assembly.AutoCycle_Running := ((#_w2 AND ("Unit1.Em6.ControlNodes".em.status.initialized OR #FALSE OR #citiTest[10]) AND #TRUE) OR "Unit1.Em6.ControlNodes".citiMap.PMC.Machining_Assembly.AutoCycle_Running) AND NOT #statUnitStatus.state.aborting AND NOT #statUnitStatus.state.stopped AND NOT #statUnitStatus.state.resetting;
END_REGION

REGION Network 95: Blocked 1
   RUNG wire#powerrail
      Contact( #FALSE )
      wire#w1
      Coil( "Unit1.Em6.ControlNodes".citiMap.PMC.Machining_Assembly.Blocked )
   END_RUNG
   RUNG wire#powerrail
      Contact( #citiTest[1] )
   END_RUNG wire#w1
   // the same network as SCL:
   "Unit1.Em6.ControlNodes".citiMap.PMC.Machining_Assembly.Blocked := #FALSE OR #citiTest[1];
END_REGION

REGION Network 96: Starved 2
   RUNG wire#powerrail
      Contact( #FALSE )
      wire#w1
      Coil( "Unit1.Em6.ControlNodes".citiMap.PMC.Machining_Assembly.Starved )
   END_RUNG
   RUNG wire#powerrail
      Contact( #citiTest[2] )
   END_RUNG wire#w1
   // the same network as SCL:
   "Unit1.Em6.ControlNodes".citiMap.PMC.Machining_Assembly.Starved := #FALSE OR #citiTest[2];
END_REGION

REGION Network 97: Good Count 3
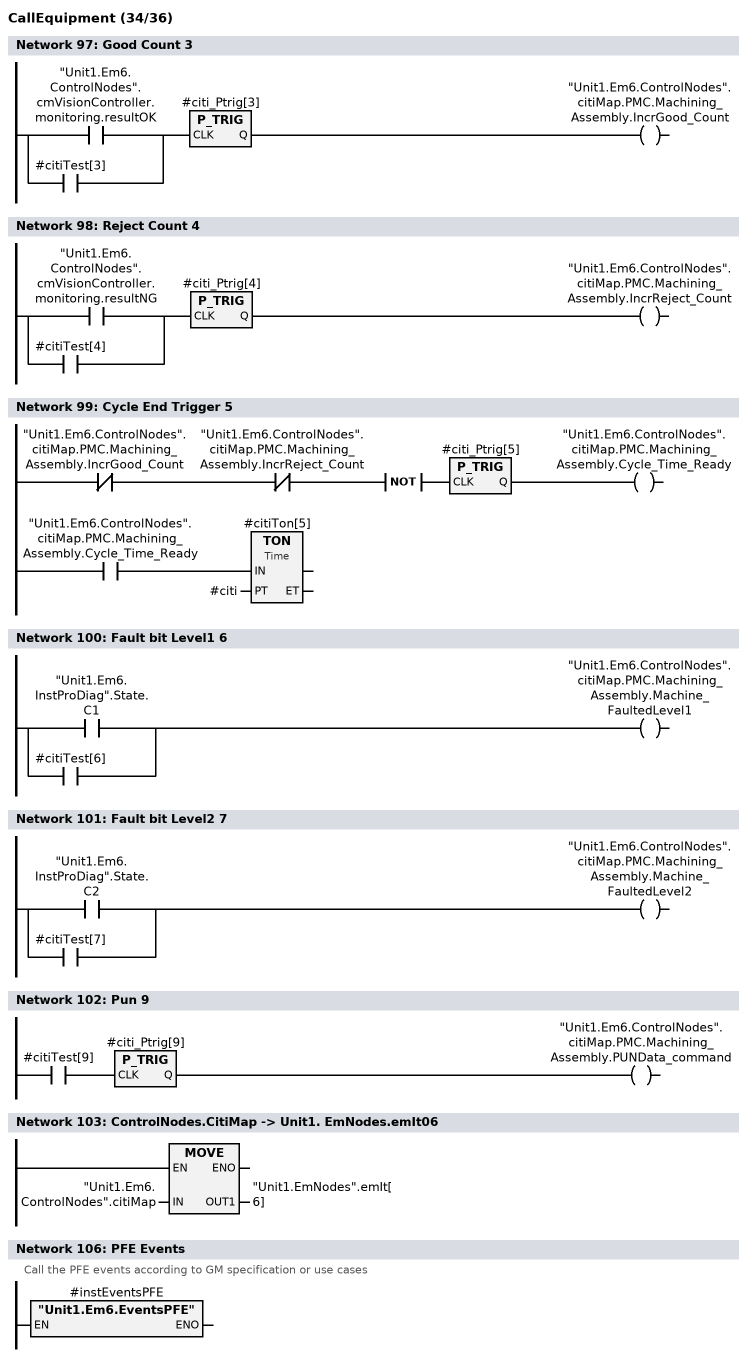
   RUNG wire#powerrail
      Contact( "Unit1.Em6.ControlNodes".cmVisionController.monitoring.resultOK )
      wire#w1
      P_Trig( #citi_Ptrig[3] )
      Coil( "Unit1.Em6.ControlNodes".citiMap.PMC.Machining_Assembly.IncrGood_Count )
   END_RUNG
   RUNG wire#powerrail
      Contact( #citiTest[3] )
   END_RUNG wire#w1
   // the same network as SCL:
   #_w1 := "Unit1.Em6.ControlNodes".cmVisionController.monitoring.resultOK OR #citiTest[3];
   #_w2 := #_w1 AND NOT #citi_Ptrig[3];   // rising edge
   #citi_Ptrig[3] := #_w1;
   "Unit1.Em6.ControlNodes".citiMap.PMC.Machining_Assembly.IncrGood_Count := #_w2;
END_REGION

REGION Network 98: Reject Count 4
   RUNG wire#powerrail
      Contact( "Unit1.Em6.ControlNodes".cmVisionController.monitoring.resultNG )
      wire#w1
      P_Trig( #citi_Ptrig[4] )
      Coil( "Unit1.Em6.ControlNodes".citiMap.PMC.Machining_Assembly.IncrReject_Count )
   END_RUNG
   RUNG wire#powerrail
      Contact( #citiTest[4] )
   END_RUNG wire#w1
   // the same network as SCL:
   #_w1 := "Unit1.Em6.ControlNodes".cmVisionController.monitoring.resultNG OR #citiTest[4];
   #_w2 := #_w1 AND NOT #citi_Ptrig[4];   // rising edge
   #citi_Ptrig[4] := #_w1;
   "Unit1.Em6.ControlNodes".citiMap.PMC.Machining_Assembly.IncrReject_Count := #_w2;
END_REGION

REGION Network 99: Cycle End Trigger 5
   RUNG wire#powerrail
      I_Contact( "Unit1.Em6.ControlNodes".citiMap.PMC.Machining_Assembly.IncrGood_Count )
      I_Contact( "Unit1.Em6.ControlNodes".citiMap.PMC.Machining_Assembly.IncrReject_Count )
      Not()
      P_Trig( #citi_Ptrig[5] )
      Coil( "Unit1.Em6.ControlNodes".citiMap.PMC.Machining_Assembly.Cycle_Time_Ready )
   END_RUNG
   RUNG wire#powerrail
      Contact( "Unit1.Em6.ControlNodes".citiMap.PMC.Machining_Assembly.Cycle_Time_Ready )
      { S7_Templates := "time_type := Time" } #citiTon[5].TON(pt := #citi, et =>)
   END_RUNG
   // the same network as SCL:
   #_w1 := NOT (NOT "Unit1.Em6.ControlNodes".citiMap.PMC.Machining_Assembly.IncrGood_Count AND NOT "Unit1.Em6.ControlNodes".citiMap.PMC.Machining_Assembly.IncrReject_Count);
   #_w2 := #_w1 AND NOT #citi_Ptrig[5];   // rising edge
   #citi_Ptrig[5] := #_w1;
   "Unit1.Em6.ControlNodes".citiMap.PMC.Machining_Assembly.Cycle_Time_Ready := #_w2;
   #citiTon[5].TON(IN := "Unit1.Em6.ControlNodes".citiMap.PMC.Machining_Assembly.Cycle_Time_Ready, PT := #citi);
END_REGION

REGION Network 100: Fault bit Level1 6
   RUNG wire#powerrail
      Contact( "Unit1.Em6.InstProDiag".State.C1 )
      wire#w1
      Coil( "Unit1.Em6.ControlNodes".citiMap.PMC.Machining_Assembly.Machine_FaultedLevel1 )
   END_RUNG
   RUNG wire#powerrail
      Contact( #citiTest[6] )
   END_RUNG wire#w1
   // the same network as SCL:
   "Unit1.Em6.ControlNodes".citiMap.PMC.Machining_Assembly.Machine_FaultedLevel1 := "Unit1.Em6.InstProDiag".State.C1 OR #citiTest[6];
END_REGION

REGION Network 101: Fault bit Level2 7
   RUNG wire#powerrail
      Contact( "Unit1.Em6.InstProDiag".State.C2 )
      wire#w1
      Coil( "Unit1.Em6.ControlNodes".citiMap.PMC.Machining_Assembly.Machine_FaultedLevel2 )
   END_RUNG
   RUNG wire#powerrail
      Contact( #citiTest[7] )
   END_RUNG wire#w1
   // the same network as SCL:
   "Unit1.Em6.ControlNodes".citiMap.PMC.Machining_Assembly.Machine_FaultedLevel2 := "Unit1.Em6.InstProDiag".State.C2 OR #citiTest[7];
END_REGION

REGION Network 102: Pun 9
   RUNG wire#powerrail
      Contact( #citiTest[9] )
      P_Trig( #citi_Ptrig[9] )
      Coil( "Unit1.Em6.ControlNodes".citiMap.PMC.Machining_Assembly.PUNData_command )
   END_RUNG
   // the same network as SCL:
   #_w1 := #citiTest[9] AND NOT #citi_Ptrig[9];   // rising edge
   #citi_Ptrig[9] := #citiTest[9];
   "Unit1.Em6.ControlNodes".citiMap.PMC.Machining_Assembly.PUNData_command := #_w1;
END_REGION

REGION Network 103: ControlNodes.CitiMap -> Unit1. EmNodes.emIt06
   RUNG wire#powerrail
      Move(in := "Unit1.Em6.ControlNodes".citiMap, out1 => "Unit1.EmNodes".emIt[6])
   END_RUNG
   // the same network as SCL:
   "Unit1.EmNodes".emIt[6] := "Unit1.Em6.ControlNodes".citiMap;
END_REGION

REGION Network 105: ******************** PFE Events ********************
END_REGION

REGION Network 106: PFE Events
   // Call the PFE events according to GM specification or use cases
   RUNG wire#powerrail
      #instEventsPFE()
   END_RUNG
   // the same network as SCL:
   #instEventsPFE();   // "Unit1.Em6.EventsPFE"
END_REGION

REGION Network 107: ******************** EM Relations Output ********************
END_REGION

REGION Network 108: EM6 Job Interface
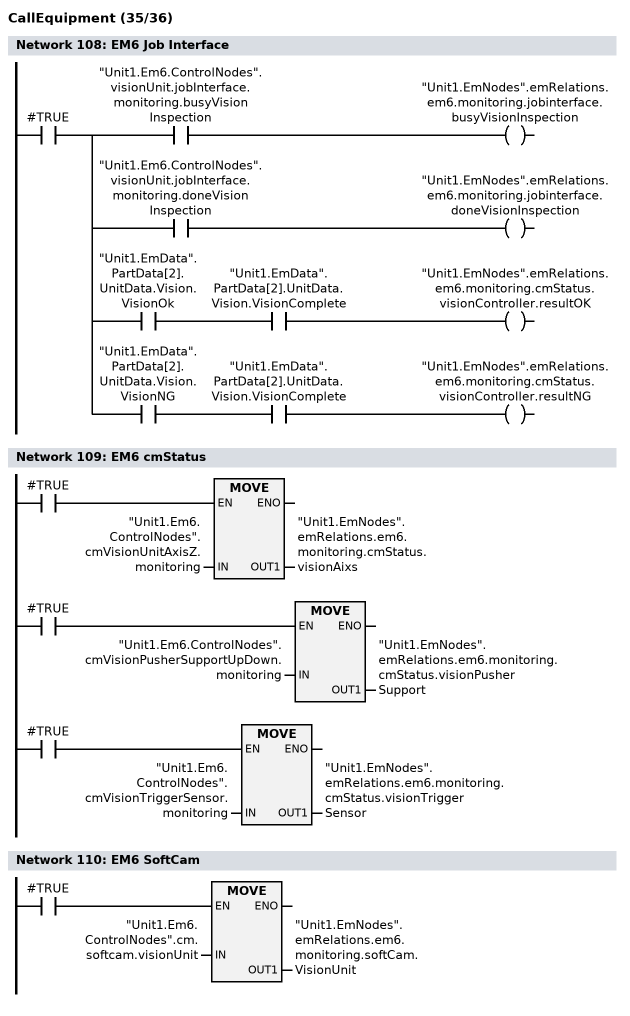
   RUNG wire#powerrail
      Contact( #TRUE )
      wire#w1
      Contact( "Unit1.Em6.ControlNodes".visionUnit.jobInterface.monitoring.busyVisionInspection )
      Coil( "Unit1.EmNodes".emRelations.em6.monitoring.jobinterface.busyVisionInspection )
   END_RUNG
   RUNG wire#w1
      Contact( "Unit1.Em6.ControlNodes".visionUnit.jobInterface.monitoring.doneVisionInspection )
      Coil( "Unit1.EmNodes".emRelations.em6.monitoring.jobinterface.doneVisionInspection )
   END_RUNG
   RUNG wire#w1
      Contact( "Unit1.EmData".PartData[2].UnitData.Vision.VisionOk )
      Contact( "Unit1.EmData".PartData[2].UnitData.Vision.VisionComplete )
      Coil( "Unit1.EmNodes".emRelations.em6.monitoring.cmStatus.visionController.resultOK )
   END_RUNG
   RUNG wire#w1
      Contact( "Unit1.EmData".PartData[2].UnitData.Vision.VisionNG )
      Contact( "Unit1.EmData".PartData[2].UnitData.Vision.VisionComplete )
      Coil( "Unit1.EmNodes".emRelations.em6.monitoring.cmStatus.visionController.resultNG )
   END_RUNG
   // the same network as SCL:
   "Unit1.EmNodes".emRelations.em6.monitoring.jobinterface.busyVisionInspection := #TRUE AND "Unit1.Em6.ControlNodes".visionUnit.jobInterface.monitoring.busyVisionInspection;
   "Unit1.EmNodes".emRelations.em6.monitoring.jobinterface.doneVisionInspection := #TRUE AND "Unit1.Em6.ControlNodes".visionUnit.jobInterface.monitoring.doneVisionInspection;
   "Unit1.EmNodes".emRelations.em6.monitoring.cmStatus.visionController.resultOK := #TRUE AND "Unit1.EmData".PartData[2].UnitData.Vision.VisionOk AND "Unit1.EmData".PartData[2].UnitData.Vision.VisionComplete;
   "Unit1.EmNodes".emRelations.em6.monitoring.cmStatus.visionController.resultNG := #TRUE AND "Unit1.EmData".PartData[2].UnitData.Vision.VisionNG AND "Unit1.EmData".PartData[2].UnitData.Vision.VisionComplete;
END_REGION

REGION Network 109: EM6 cmStatus
   RUNG wire#powerrail
      Contact( #TRUE )
      { S7_GenerateENO := "TRUE" } Move(in := "Unit1.Em6.ControlNodes".cmVisionUnitAxisZ.monitoring, out1 => "Unit1.EmNodes".emRelations.em6.monitoring.cmStatus.visionAixs)
   END_RUNG
   RUNG wire#powerrail
      Contact( #TRUE )
      { S7_GenerateENO := "TRUE" } Move(in := "Unit1.Em6.ControlNodes".cmVisionPusherSupportUpDown.monitoring, out1 => "Unit1.EmNodes".emRelations.em6.monitoring.cmStatus.visionPusherSupport)
   END_RUNG
   RUNG wire#powerrail
      Contact( #TRUE )
      { S7_GenerateENO := "TRUE" } Move(in := "Unit1.Em6.ControlNodes".cmVisionTriggerSensor.monitoring, out1 => "Unit1.EmNodes".emRelations.em6.monitoring.cmStatus.visionTriggerSensor)
   END_RUNG
   // the same network as SCL:
   IF #TRUE THEN
       "Unit1.EmNodes".emRelations.em6.monitoring.cmStatus.visionAixs := "Unit1.Em6.ControlNodes".cmVisionUnitAxisZ.monitoring;
       "Unit1.EmNodes".emRelations.em6.monitoring.cmStatus.visionPusherSupport := "Unit1.Em6.ControlNodes".cmVisionPusherSupportUpDown.monitoring;
       "Unit1.EmNodes".emRelations.em6.monitoring.cmStatus.visionTriggerSensor := "Unit1.Em6.ControlNodes".cmVisionTriggerSensor.monitoring;
   END_IF;
END_REGION

REGION Network 110: EM6 SoftCam
   RUNG wire#powerrail
      Contact( #TRUE )
      { S7_GenerateENO := "TRUE" } Move(in := "Unit1.Em6.ControlNodes".cm.softcam.visionUnit, out1 => "Unit1.EmNodes".emRelations.em6.monitoring.softCam.VisionUnit)
   END_RUNG
   // the same network as SCL:
   IF #TRUE THEN
       "Unit1.EmNodes".emRelations.em6.monitoring.softCam.VisionUnit := "Unit1.Em6.ControlNodes".cm.softcam.visionUnit;
   END_IF;
END_REGION

REGION Network 111: EM6 UserDefine
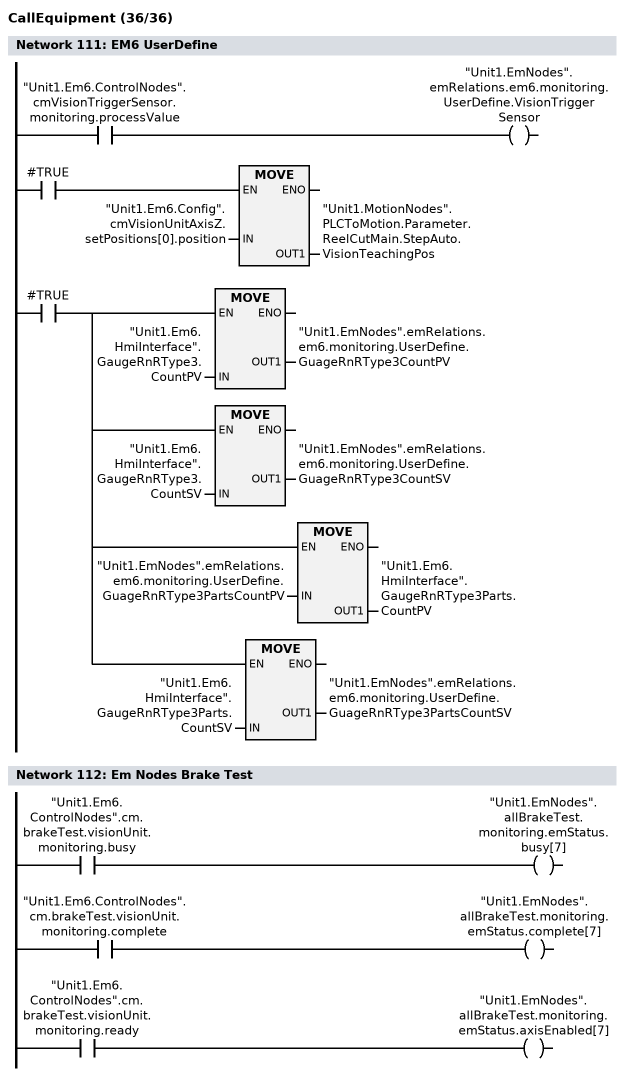
   RUNG wire#powerrail
      Contact( "Unit1.Em6.ControlNodes".cmVisionTriggerSensor.monitoring.processValue )
      Coil( "Unit1.EmNodes".emRelations.em6.monitoring.UserDefine.VisionTriggerSensor )
   END_RUNG
   RUNG wire#powerrail
      Contact( #TRUE )
      Move(in := "Unit1.Em6.Config".cmVisionUnitAxisZ.setPositions[0].position, out1 => "Unit1.MotionNodes".PLCToMotion.Parameter.ReelCutMain.StepAuto.VisionTeachingPos)
   END_RUNG
   RUNG wire#powerrail
      Contact( #TRUE )
      wire#w1
      Move(in := "Unit1.Em6.HmiInterface".GaugeRnRType3.CountPV, out1 => "Unit1.EmNodes".emRelations.em6.monitoring.UserDefine.GuageRnRType3CountPV)
   END_RUNG
   RUNG wire#w1
      Move(in := "Unit1.Em6.HmiInterface".GaugeRnRType3.CountSV, out1 => "Unit1.EmNodes".emRelations.em6.monitoring.UserDefine.GuageRnRType3CountSV)
   END_RUNG
   RUNG wire#w1
      Move(in := "Unit1.EmNodes".emRelations.em6.monitoring.UserDefine.GuageRnRType3PartsCountPV, out1 => "Unit1.Em6.HmiInterface".GaugeRnRType3Parts.CountPV)
   END_RUNG
   RUNG wire#w1
      Move(in := "Unit1.Em6.HmiInterface".GaugeRnRType3Parts.CountSV, out1 => "Unit1.EmNodes".emRelations.em6.monitoring.UserDefine.GuageRnRType3PartsCountSV)
   END_RUNG
   // the same network as SCL:
   "Unit1.EmNodes".emRelations.em6.monitoring.UserDefine.VisionTriggerSensor := "Unit1.Em6.ControlNodes".cmVisionTriggerSensor.monitoring.processValue;
   IF #TRUE THEN
       "Unit1.MotionNodes".PLCToMotion.Parameter.ReelCutMain.StepAuto.VisionTeachingPos := "Unit1.Em6.Config".cmVisionUnitAxisZ.setPositions[0].position;
       "Unit1.EmNodes".emRelations.em6.monitoring.UserDefine.GuageRnRType3CountPV := "Unit1.Em6.HmiInterface".GaugeRnRType3.CountPV;
       "Unit1.EmNodes".emRelations.em6.monitoring.UserDefine.GuageRnRType3CountSV := "Unit1.Em6.HmiInterface".GaugeRnRType3.CountSV;
       "Unit1.Em6.HmiInterface".GaugeRnRType3Parts.CountPV := "Unit1.EmNodes".emRelations.em6.monitoring.UserDefine.GuageRnRType3PartsCountPV;
       "Unit1.EmNodes".emRelations.em6.monitoring.UserDefine.GuageRnRType3PartsCountSV := "Unit1.Em6.HmiInterface".GaugeRnRType3Parts.CountSV;
   END_IF;
END_REGION

REGION Network 112: Em Nodes Brake Test
   RUNG wire#powerrail
      Contact( "Unit1.Em6.ControlNodes".cm.brakeTest.visionUnit.monitoring.busy )
      Coil( "Unit1.EmNodes".allBrakeTest.monitoring.emStatus.busy[7] )
   END_RUNG
   RUNG wire#powerrail
      Contact( "Unit1.Em6.ControlNodes".cm.brakeTest.visionUnit.monitoring.complete )
      Coil( "Unit1.EmNodes".allBrakeTest.monitoring.emStatus.complete[7] )
   END_RUNG
   RUNG wire#powerrail
      Contact( "Unit1.Em6.ControlNodes".cm.brakeTest.visionUnit.monitoring.ready )
      Coil( "Unit1.EmNodes".allBrakeTest.monitoring.emStatus.axisEnabled[7] )
   END_RUNG
   // the same network as SCL:
   "Unit1.EmNodes".allBrakeTest.monitoring.emStatus.busy[7] := "Unit1.Em6.ControlNodes".cm.brakeTest.visionUnit.monitoring.busy;
   "Unit1.EmNodes".allBrakeTest.monitoring.emStatus.complete[7] := "Unit1.Em6.ControlNodes".cm.brakeTest.visionUnit.monitoring.complete;
   "Unit1.EmNodes".allBrakeTest.monitoring.emStatus.axisEnabled[7] := "Unit1.Em6.ControlNodes".cm.brakeTest.visionUnit.monitoring.ready;
END_REGION
END_FUNCTION_BLOCK
